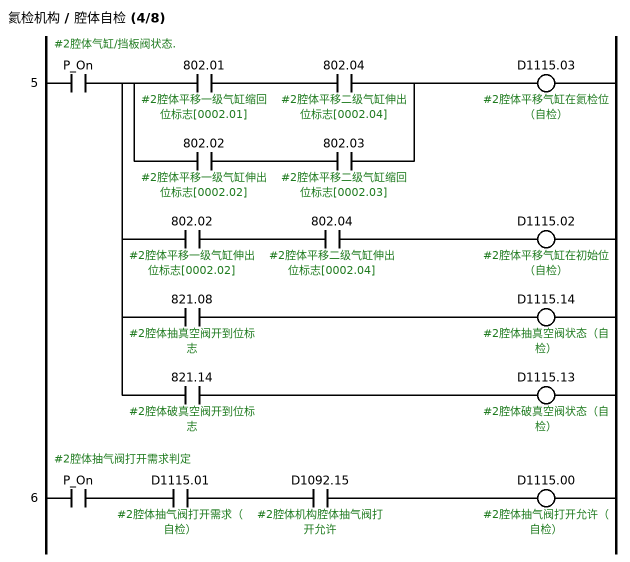
; rung 5: #2腔体气缸/挡板阀状态.
LD P_On
OUT TR0
LD 802.01  ; #2腔体平移一级气缸缩回位标志[0002.01]
AND 802.04  ; #2腔体平移二级气缸伸出位标志[0002.04]
LD 802.02  ; #2腔体平移一级气缸伸出位标志[0002.02]
AND 802.03  ; #2腔体平移二级气缸缩回位标志[0002.03]
ORLD
ANDLD
OUT D1115.03  ; #2腔体平移气缸在氦检位（自检）
LD TR0
AND 802.02  ; #2腔体平移一级气缸伸出位标志[0002.02]
AND 802.04  ; #2腔体平移二级气缸伸出位标志[0002.04]
OUT D1115.02  ; #2腔体平移气缸在初始位（自检）
LD TR0
AND 821.08  ; #2腔体抽真空阀开到位标志
OUT D1115.14  ; #2腔体抽真空阀状态（自检）
LD TR0
AND 821.14  ; #2腔体破真空阀开到位标志
OUT D1115.13  ; #2腔体破真空阀状态（自检）
; rung 6: #2腔体抽气阀打开需求判定
LD P_On
AND D1115.01  ; #2腔体抽气阀打开需求（自检）
AND D1092.15  ; #2腔体机构腔体抽气阀打开允许
OUT D1115.00  ; #2腔体抽气阀打开允许（自检）

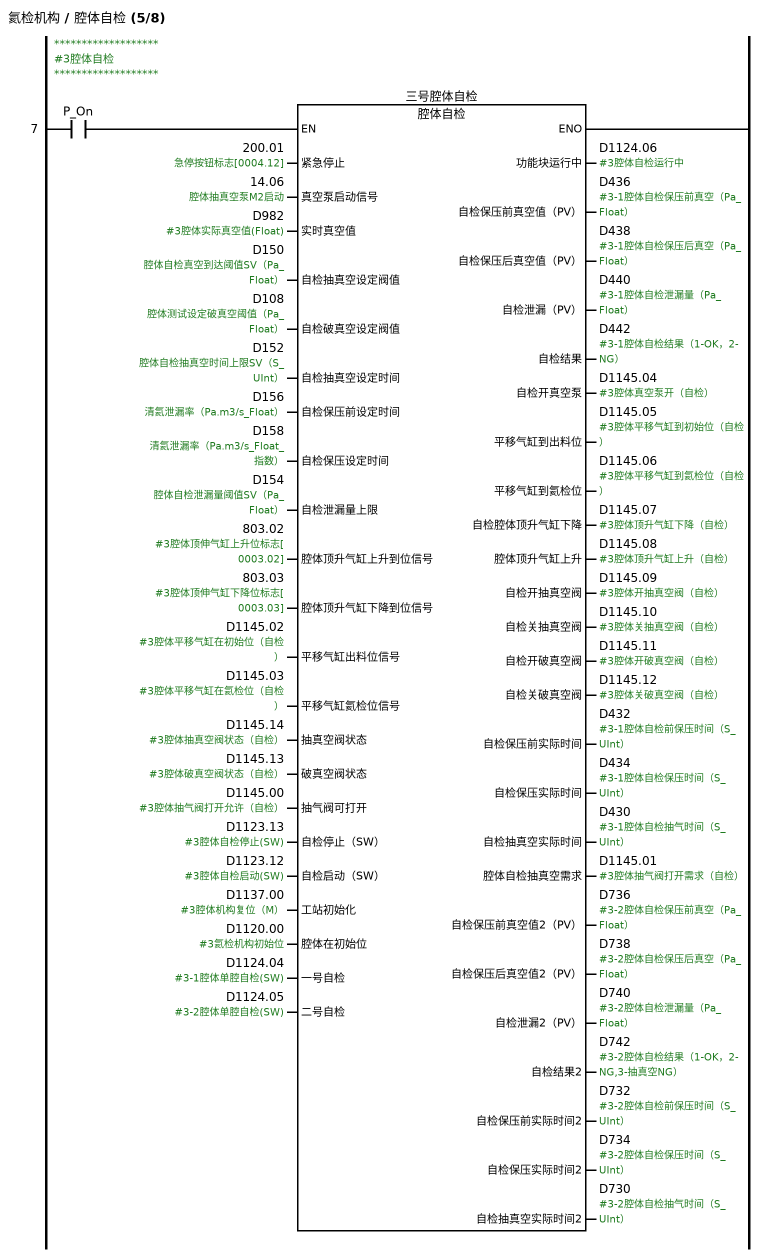
; rung 7: ******************* / #3腔体自检 / *******************
LD P_On
CALL 三号腔体自检 : 腔体自检 (紧急停止 := 200.01, 真空泵启动信号 := 14.06, 实时真空值 := D982, 自检抽真空设定阀值 := D150, 自检破真空设定阀值 := D108, 自检抽真空设定时间 := D152, 自检保压前设定时间 := D156, 自检保压设定时间 := D158, 自检泄漏量上限 := D154, 腔体顶升气缸上升到位信号 := 803.02, 腔体顶升气缸下降到位信号 := 803.03, 平移气缸出料位信号 := D1145.02, 平移气缸氦检位信号 := D1145.03, 抽真空阀状态 := D1145.14, 破真空阀状态 := D1145.13, 抽气阀可打开 := D1145.00, 自检停止（SW） := D1123.13, 自检启动（SW） := D1123.12, 工站初始化 := D1137.00, 腔体在初始位 := D1120.00, 一号自检 := D1124.04, 二号自检 := D1124.05, 功能块运行中 => D1124.06, 自检保压前真空值（PV） => D436, 自检保压后真空值（PV） => D438, 自检泄漏（PV） => D440, 自检结果 => D442, 自检开真空泵 => D1145.04, 平移气缸到出料位 => D1145.05, 平移气缸到氦检位 => D1145.06, 自检腔体顶升气缸下降 => D1145.07, 腔体顶升气缸上升 => D1145.08, 自检开抽真空阀 => D1145.09, 自检关抽真空阀 => D1145.10, 自检开破真空阀 => D1145.11, 自检关破真空阀 => D1145.12, 自检保压前实际时间 => D432, 自检保压实际时间 => D434, 自检抽真空实际时间 => D430, 腔体自检抽真空需求 => D1145.01, 自检保压前真空值2（PV） => D736, 自检保压后真空值2（PV） => D738, 自检泄漏2（PV） => D740, 自检结果2 => D742, 自检保压前实际时间2 => D732, 自检保压实际时间2 => D734, 自检抽真空实际时间2 => D730)  ; 急停按钮标志[0004.12], 腔体抽真空泵M2启动, #3腔体实际真空值(Float), 腔体自检真空到达阈值SV（Pa_Float）, 腔体测试设定破真空阈值（Pa_Float）, 腔体自检抽真空时间上限SV（S_UInt）, 清氦泄漏率（Pa.m3/s_Float）, 清氦泄漏率（Pa.m3/s_Float_指数）, 腔体自检泄漏量阈值SV（Pa_Float）, #3腔体顶伸气缸上升位标志[0003.02], #3腔体顶伸气缸下降位标志[0003.03], #3腔体平移气缸在初始位（自检）, #3腔体平移气缸在氦检位（自检）, #3腔体抽真空阀状态（自检）, #3腔体破真空阀状态（自检）, #3腔体抽气阀打开允许（自检）, #3腔体自检停止(SW), #3腔体自检启动(SW), #3腔体机构复位（M）, #3氦检机构初始位, #3-1腔体单腔自检(SW), #3-2腔体单腔自检(SW), #3腔体自检运行中, #3-1腔体自检保压前真空（Pa_Float）, #3-1腔体自检保压后真空（Pa_Float）, #3-1腔体自检泄漏量（Pa_Float）, #3-1腔体自检结果（1-OK，2-NG）, #3腔体真空泵开（自检）, #3腔体平移气缸到初始位（自检）, #3腔体平移气缸到氦检位（自检）, #3腔体顶升气缸下降（自检）, #3腔体顶升气缸上升（自检）, #3腔体开抽真空阀（自检）, #3腔体关抽真空阀（自检）, #3腔体开破真空阀（自检）, #3腔体关破真空阀（自检）, #3-1腔体自检前保压时间（S_UInt）, #3-1腔体自检保压时间（S_UInt）, #3-1腔体自检抽气时间（S_UInt）, #3腔体抽气阀打开需求（自检）, #3-2腔体自检保压前真空（Pa_Float）, #3-2腔体自检保压后真空（Pa_Float）, #3-2腔体自检泄漏量（Pa_Float）, #3-2腔体自检结果（1-OK，2-NG,3-抽真空NG）, #3-2腔体自检前保压时间（S_UInt）, #3-2腔体自检保压时间（S_UInt）, #3-2腔体自检抽气时间（S_UInt）

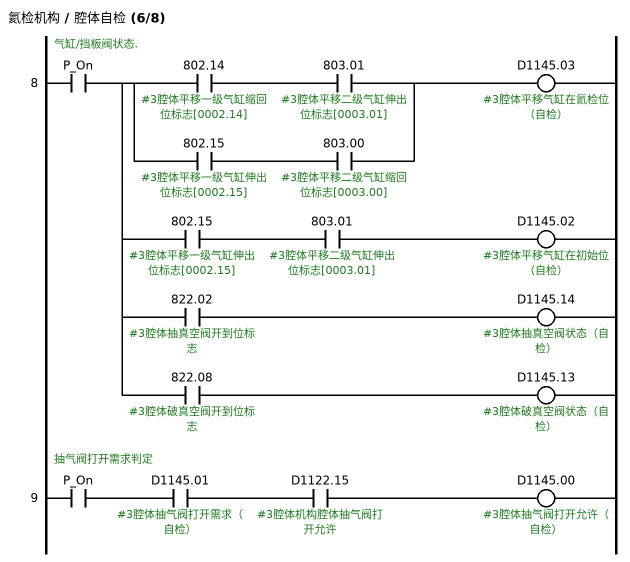
; rung 8: 气缸/挡板阀状态.
LD P_On
OUT TR0
LD 802.14  ; #3腔体平移一级气缸缩回位标志[0002.14]
AND 803.01  ; #3腔体平移二级气缸伸出位标志[0003.01]
LD 802.15  ; #3腔体平移一级气缸伸出位标志[0002.15]
AND 803.00  ; #3腔体平移二级气缸缩回位标志[0003.00]
ORLD
ANDLD
OUT D1145.03  ; #3腔体平移气缸在氦检位（自检）
LD TR0
AND 802.15  ; #3腔体平移一级气缸伸出位标志[0002.15]
AND 803.01  ; #3腔体平移二级气缸伸出位标志[0003.01]
OUT D1145.02  ; #3腔体平移气缸在初始位（自检）
LD TR0
AND 822.02  ; #3腔体抽真空阀开到位标志
OUT D1145.14  ; #3腔体抽真空阀状态（自检）
LD TR0
AND 822.08  ; #3腔体破真空阀开到位标志
OUT D1145.13  ; #3腔体破真空阀状态（自检）
; rung 9: 抽气阀打开需求判定
LD P_On
AND D1145.01  ; #3腔体抽气阀打开需求（自检）
AND D1122.15  ; #3腔体机构腔体抽气阀打开允许
OUT D1145.00  ; #3腔体抽气阀打开允许（自检）

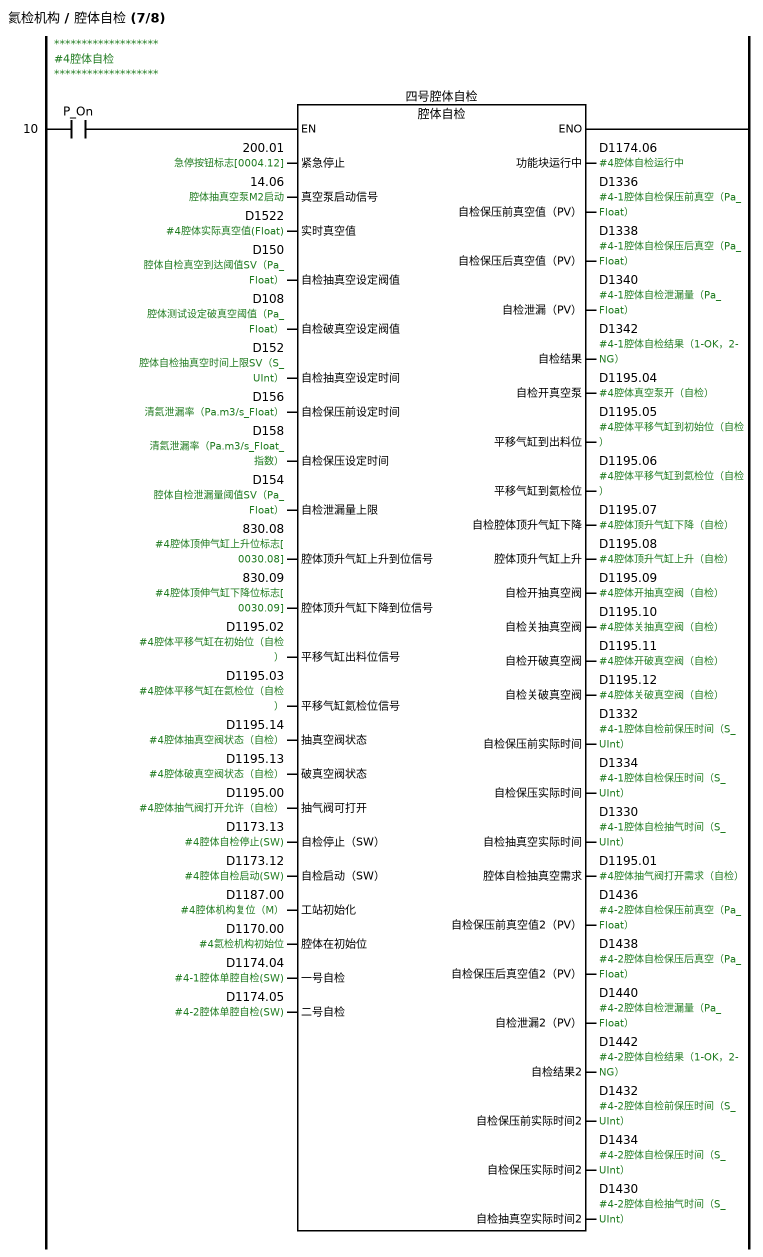
; rung 10: ******************* / #4腔体自检 / *******************
LD P_On
CALL 四号腔体自检 : 腔体自检 (紧急停止 := 200.01, 真空泵启动信号 := 14.06, 实时真空值 := D1522, 自检抽真空设定阀值 := D150, 自检破真空设定阀值 := D108, 自检抽真空设定时间 := D152, 自检保压前设定时间 := D156, 自检保压设定时间 := D158, 自检泄漏量上限 := D154, 腔体顶升气缸上升到位信号 := 830.08, 腔体顶升气缸下降到位信号 := 830.09, 平移气缸出料位信号 := D1195.02, 平移气缸氦检位信号 := D1195.03, 抽真空阀状态 := D1195.14, 破真空阀状态 := D1195.13, 抽气阀可打开 := D1195.00, 自检停止（SW） := D1173.13, 自检启动（SW） := D1173.12, 工站初始化 := D1187.00, 腔体在初始位 := D1170.00, 一号自检 := D1174.04, 二号自检 := D1174.05, 功能块运行中 => D1174.06, 自检保压前真空值（PV） => D1336, 自检保压后真空值（PV） => D1338, 自检泄漏（PV） => D1340, 自检结果 => D1342, 自检开真空泵 => D1195.04, 平移气缸到出料位 => D1195.05, 平移气缸到氦检位 => D1195.06, 自检腔体顶升气缸下降 => D1195.07, 腔体顶升气缸上升 => D1195.08, 自检开抽真空阀 => D1195.09, 自检关抽真空阀 => D1195.10, 自检开破真空阀 => D1195.11, 自检关破真空阀 => D1195.12, 自检保压前实际时间 => D1332, 自检保压实际时间 => D1334, 自检抽真空实际时间 => D1330, 腔体自检抽真空需求 => D1195.01, 自检保压前真空值2（PV） => D1436, 自检保压后真空值2（PV） => D1438, 自检泄漏2（PV） => D1440, 自检结果2 => D1442, 自检保压前实际时间2 => D1432, 自检保压实际时间2 => D1434, 自检抽真空实际时间2 => D1430)  ; 急停按钮标志[0004.12], 腔体抽真空泵M2启动, #4腔体实际真空值(Float), 腔体自检真空到达阈值SV（Pa_Float）, 腔体测试设定破真空阈值（Pa_Float）, 腔体自检抽真空时间上限SV（S_UInt）, 清氦泄漏率（Pa.m3/s_Float）, 清氦泄漏率（Pa.m3/s_Float_指数）, 腔体自检泄漏量阈值SV（Pa_Float）, #4腔体顶伸气缸上升位标志[0030.08], #4腔体顶伸气缸下降位标志[0030.09], #4腔体平移气缸在初始位（自检）, #4腔体平移气缸在氦检位（自检）, #4腔体抽真空阀状态（自检）, #4腔体破真空阀状态（自检）, #4腔体抽气阀打开允许（自检）, #4腔体自检停止(SW), #4腔体自检启动(SW), #4腔体机构复位（M）, #4氦检机构初始位, #4-1腔体单腔自检(SW), #4-2腔体单腔自检(SW), #4腔体自检运行中, #4-1腔体自检保压前真空（Pa_Float）, #4-1腔体自检保压后真空（Pa_Float）, #4-1腔体自检泄漏量（Pa_Float）, #4-1腔体自检结果（1-OK，2-NG）, #4腔体真空泵开（自检）, #4腔体平移气缸到初始位（自检）, #4腔体平移气缸到氦检位（自检）, #4腔体顶升气缸下降（自检）, #4腔体顶升气缸上升（自检）, #4腔体开抽真空阀（自检）, #4腔体关抽真空阀（自检）, #4腔体开破真空阀（自检）, #4腔体关破真空阀（自检）, #4-1腔体自检前保压时间（S_UInt）, #4-1腔体自检保压时间（S_UInt）, #4-1腔体自检抽气时间（S_UInt）, #4腔体抽气阀打开需求（自检）, #4-2腔体自检保压前真空（Pa_Float）, #4-2腔体自检保压后真空（Pa_Float）, #4-2腔体自检泄漏量（Pa_Float）, #4-2腔体自检结果（1-OK，2-NG）, #4-2腔体自检前保压时间（S_UInt）, #4-2腔体自检保压时间（S_UInt）, #4-2腔体自检抽气时间（S_UInt）

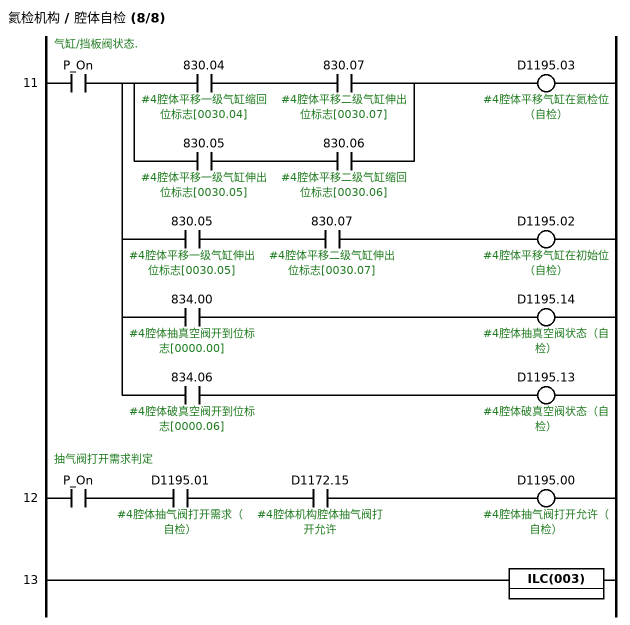
; rung 11: 气缸/挡板阀状态.
LD P_On
OUT TR0
LD 830.04  ; #4腔体平移一级气缸缩回位标志[0030.04]
AND 830.07  ; #4腔体平移二级气缸伸出位标志[0030.07]
LD 830.05  ; #4腔体平移一级气缸伸出位标志[0030.05]
AND 830.06  ; #4腔体平移二级气缸缩回位标志[0030.06]
ORLD
ANDLD
OUT D1195.03  ; #4腔体平移气缸在氦检位（自检）
LD TR0
AND 830.05  ; #4腔体平移一级气缸伸出位标志[0030.05]
AND 830.07  ; #4腔体平移二级气缸伸出位标志[0030.07]
OUT D1195.02  ; #4腔体平移气缸在初始位（自检）
LD TR0
AND 834.00  ; #4腔体抽真空阀开到位标志[0000.00]
OUT D1195.14  ; #4腔体抽真空阀状态（自检）
LD TR0
AND 834.06  ; #4腔体破真空阀开到位标志[0000.06]
OUT D1195.13  ; #4腔体破真空阀状态（自检）
; rung 12: 抽气阀打开需求判定
LD P_On
AND D1195.01  ; #4腔体抽气阀打开需求（自检）
AND D1172.15  ; #4腔体机构腔体抽气阀打开允许
OUT D1195.00  ; #4腔体抽气阀打开允许（自检）
; rung 13
ILC(003)

### Section 指示灯

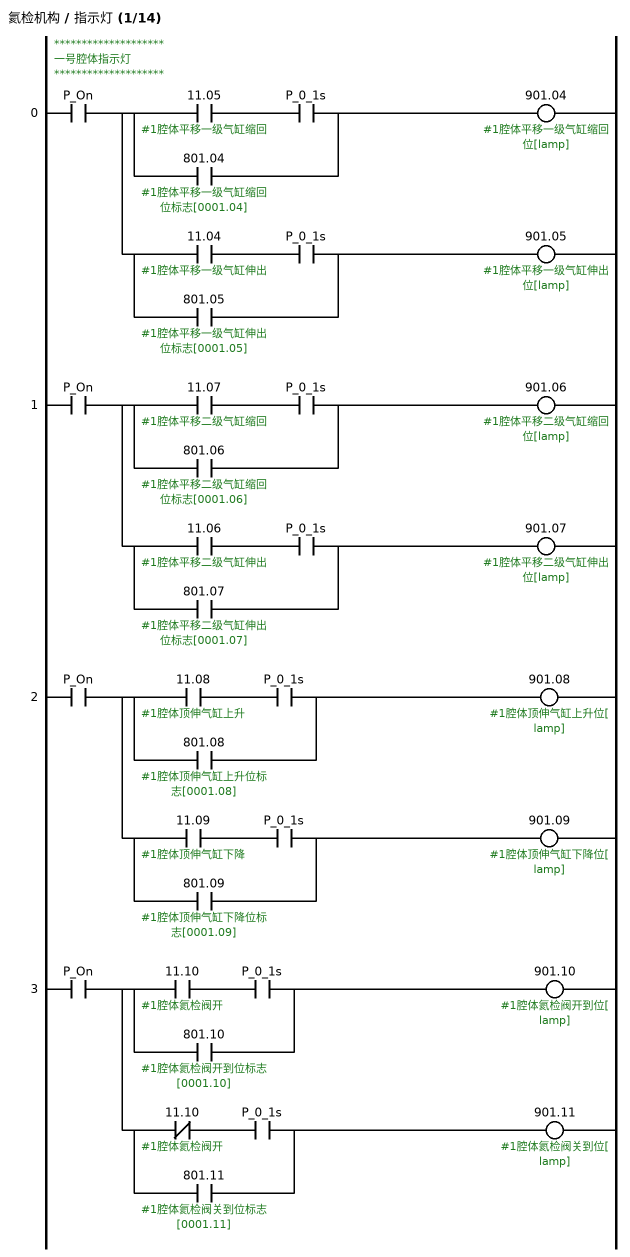
; rung 0: ******************** / 一号腔体指示灯 / ********************
LD P_On
OUT TR0
LD 11.05  ; #1腔体平移一级气缸缩回
AND P_0_1s
OR 801.04  ; #1腔体平移一级气缸缩回位标志[0001.04]
ANDLD
OUT 901.04  ; #1腔体平移一级气缸缩回位[lamp]
LD TR0
LD 11.04  ; #1腔体平移一级气缸伸出
AND P_0_1s
OR 801.05  ; #1腔体平移一级气缸伸出位标志[0001.05]
ANDLD
OUT 901.05  ; #1腔体平移一级气缸伸出位[lamp]
; rung 1
LD P_On
OUT TR0
LD 11.07  ; #1腔体平移二级气缸缩回
AND P_0_1s
OR 801.06  ; #1腔体平移二级气缸缩回位标志[0001.06]
ANDLD
OUT 901.06  ; #1腔体平移二级气缸缩回位[lamp]
LD TR0
LD 11.06  ; #1腔体平移二级气缸伸出
AND P_0_1s
OR 801.07  ; #1腔体平移二级气缸伸出位标志[0001.07]
ANDLD
OUT 901.07  ; #1腔体平移二级气缸伸出位[lamp]
; rung 2
LD P_On
OUT TR0
LD 11.08  ; #1腔体顶伸气缸上升
AND P_0_1s
OR 801.08  ; #1腔体顶伸气缸上升位标志[0001.08]
ANDLD
OUT 901.08  ; #1腔体顶伸气缸上升位[lamp]
LD TR0
LD 11.09  ; #1腔体顶伸气缸下降
AND P_0_1s
OR 801.09  ; #1腔体顶伸气缸下降位标志[0001.09]
ANDLD
OUT 901.09  ; #1腔体顶伸气缸下降位[lamp]
; rung 3
LD P_On
OUT TR0
LD 11.10  ; #1腔体氦检阀开
AND P_0_1s
OR 801.10  ; #1腔体氦检阀开到位标志[0001.10]
ANDLD
OUT 901.10  ; #1腔体氦检阀开到位[lamp]
LD TR0
LDNOT 11.10  ; #1腔体氦检阀开
AND P_0_1s
OR 801.11  ; #1腔体氦检阀关到位标志[0001.11]
ANDLD
OUT 901.11  ; #1腔体氦检阀关到位[lamp]

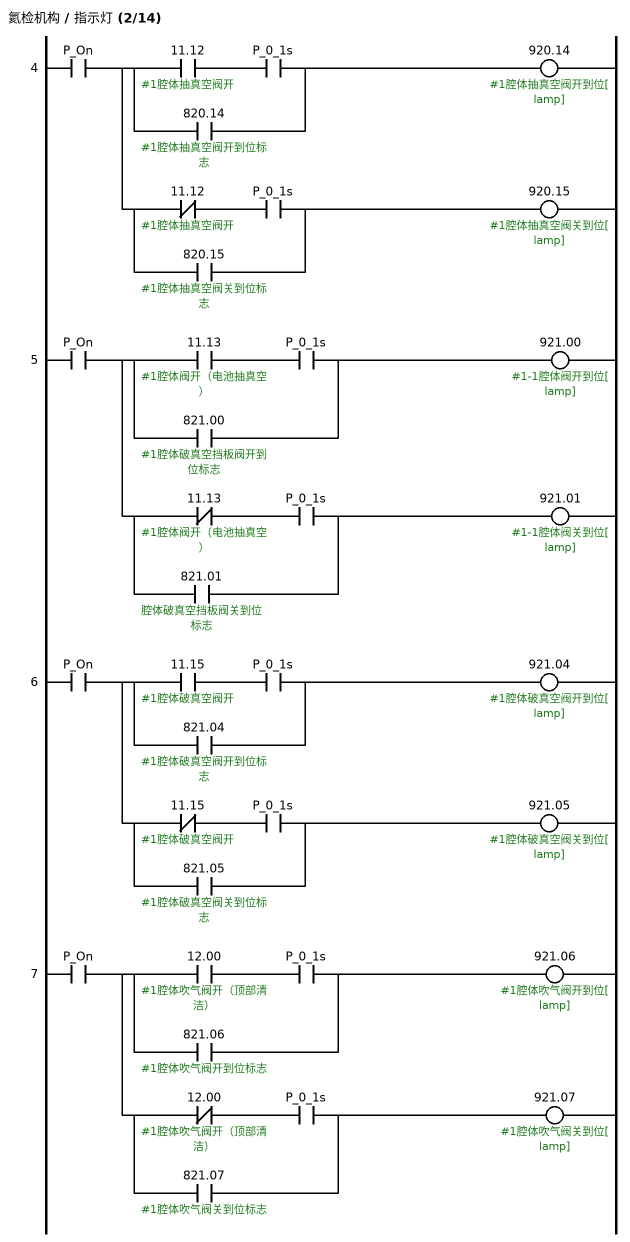
; rung 4
LD P_On
OUT TR0
LD 11.12  ; #1腔体抽真空阀开
AND P_0_1s
OR 820.14  ; #1腔体抽真空阀开到位标志
ANDLD
OUT 920.14  ; #1腔体抽真空阀开到位[lamp]
LD TR0
LDNOT 11.12  ; #1腔体抽真空阀开
AND P_0_1s
OR 820.15  ; #1腔体抽真空阀关到位标志
ANDLD
OUT 920.15  ; #1腔体抽真空阀关到位[lamp]
; rung 5
LD P_On
OUT TR0
LD 11.13  ; #1腔体阀开（电池抽真空）
AND P_0_1s
OR 821.00  ; #1腔体破真空挡板阀开到位标志
ANDLD
OUT 921.00  ; #1-1腔体阀开到位[lamp]
LD TR0
LDNOT 11.13  ; #1腔体阀开（电池抽真空）
AND P_0_1s
OR 821.01  ; 腔体破真空挡板阀关到位标志
ANDLD
OUT 921.01  ; #1-1腔体阀关到位[lamp]
; rung 6
LD P_On
OUT TR0
LD 11.15  ; #1腔体破真空阀开
AND P_0_1s
OR 821.04  ; #1腔体破真空阀开到位标志
ANDLD
OUT 921.04  ; #1腔体破真空阀开到位[lamp]
LD TR0
LDNOT 11.15  ; #1腔体破真空阀开
AND P_0_1s
OR 821.05  ; #1腔体破真空阀关到位标志
ANDLD
OUT 921.05  ; #1腔体破真空阀关到位[lamp]
; rung 7
LD P_On
OUT TR0
LD 12.00  ; #1腔体吹气阀开（顶部清洁）
AND P_0_1s
OR 821.06  ; #1腔体吹气阀开到位标志
ANDLD
OUT 921.06  ; #1腔体吹气阀开到位[lamp]
LD TR0
LDNOT 12.00  ; #1腔体吹气阀开（顶部清洁）
AND P_0_1s
OR 821.07  ; #1腔体吹气阀关到位标志
ANDLD
OUT 921.07  ; #1腔体吹气阀关到位[lamp]

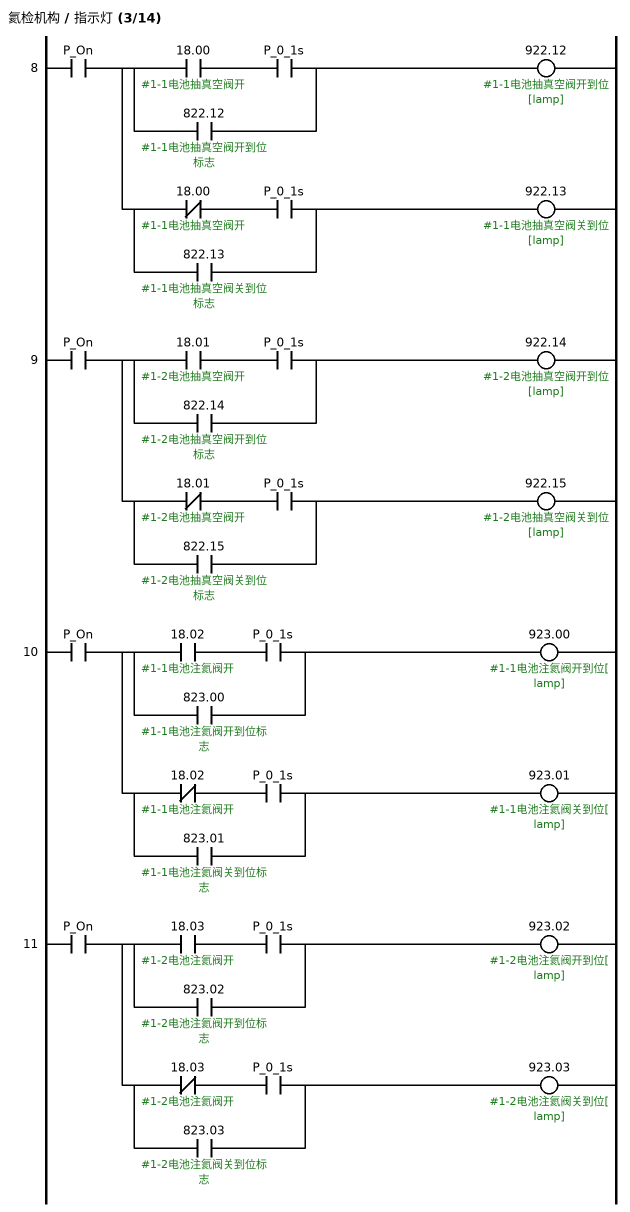
; rung 8
LD P_On
OUT TR0
LD 18.00  ; #1-1电池抽真空阀开
AND P_0_1s
OR 822.12  ; #1-1电池抽真空阀开到位标志
ANDLD
OUT 922.12  ; #1-1电池抽真空阀开到位[lamp]
LD TR0
LDNOT 18.00  ; #1-1电池抽真空阀开
AND P_0_1s
OR 822.13  ; #1-1电池抽真空阀关到位标志
ANDLD
OUT 922.13  ; #1-1电池抽真空阀关到位[lamp]
; rung 9
LD P_On
OUT TR0
LD 18.01  ; #1-2电池抽真空阀开
AND P_0_1s
OR 822.14  ; #1-2电池抽真空阀开到位标志
ANDLD
OUT 922.14  ; #1-2电池抽真空阀开到位[lamp]
LD TR0
LDNOT 18.01  ; #1-2电池抽真空阀开
AND P_0_1s
OR 822.15  ; #1-2电池抽真空阀关到位标志
ANDLD
OUT 922.15  ; #1-2电池抽真空阀关到位[lamp]
; rung 10
LD P_On
OUT TR0
LD 18.02  ; #1-1电池注氦阀开
AND P_0_1s
OR 823.00  ; #1-1电池注氦阀开到位标志
ANDLD
OUT 923.00  ; #1-1电池注氦阀开到位[lamp]
LD TR0
LDNOT 18.02  ; #1-1电池注氦阀开
AND P_0_1s
OR 823.01  ; #1-1电池注氦阀关到位标志
ANDLD
OUT 923.01  ; #1-1电池注氦阀关到位[lamp]
; rung 11
LD P_On
OUT TR0
LD 18.03  ; #1-2电池注氦阀开
AND P_0_1s
OR 823.02  ; #1-2电池注氦阀开到位标志
ANDLD
OUT 923.02  ; #1-2电池注氦阀开到位[lamp]
LD TR0
LDNOT 18.03  ; #1-2电池注氦阀开
AND P_0_1s
OR 823.03  ; #1-2电池注氦阀关到位标志
ANDLD
OUT 923.03  ; #1-2电池注氦阀关到位[lamp]

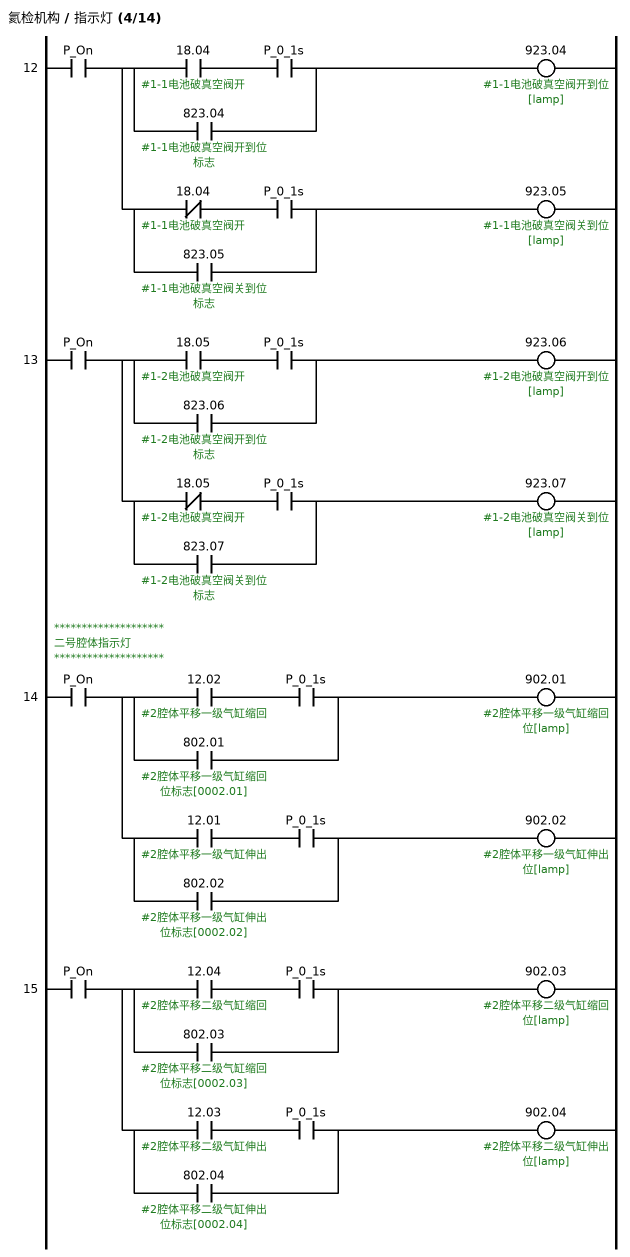
; rung 12
LD P_On
OUT TR0
LD 18.04  ; #1-1电池破真空阀开
AND P_0_1s
OR 823.04  ; #1-1电池破真空阀开到位标志
ANDLD
OUT 923.04  ; #1-1电池破真空阀开到位[lamp]
LD TR0
LDNOT 18.04  ; #1-1电池破真空阀开
AND P_0_1s
OR 823.05  ; #1-1电池破真空阀关到位标志
ANDLD
OUT 923.05  ; #1-1电池破真空阀关到位[lamp]
; rung 13
LD P_On
OUT TR0
LD 18.05  ; #1-2电池破真空阀开
AND P_0_1s
OR 823.06  ; #1-2电池破真空阀开到位标志
ANDLD
OUT 923.06  ; #1-2电池破真空阀开到位[lamp]
LD TR0
LDNOT 18.05  ; #1-2电池破真空阀开
AND P_0_1s
OR 823.07  ; #1-2电池破真空阀关到位标志
ANDLD
OUT 923.07  ; #1-2电池破真空阀关到位[lamp]
; rung 14: ******************** / 二号腔体指示灯 / ********************
LD P_On
OUT TR0
LD 12.02  ; #2腔体平移一级气缸缩回
AND P_0_1s
OR 802.01  ; #2腔体平移一级气缸缩回位标志[0002.01]
ANDLD
OUT 902.01  ; #2腔体平移一级气缸缩回位[lamp]
LD TR0
LD 12.01  ; #2腔体平移一级气缸伸出
AND P_0_1s
OR 802.02  ; #2腔体平移一级气缸伸出位标志[0002.02]
ANDLD
OUT 902.02  ; #2腔体平移一级气缸伸出位[lamp]
; rung 15
LD P_On
OUT TR0
LD 12.04  ; #2腔体平移二级气缸缩回
AND P_0_1s
OR 802.03  ; #2腔体平移二级气缸缩回位标志[0002.03]
ANDLD
OUT 902.03  ; #2腔体平移二级气缸缩回位[lamp]
LD TR0
LD 12.03  ; #2腔体平移二级气缸伸出
AND P_0_1s
OR 802.04  ; #2腔体平移二级气缸伸出位标志[0002.04]
ANDLD
OUT 902.04  ; #2腔体平移二级气缸伸出位[lamp]

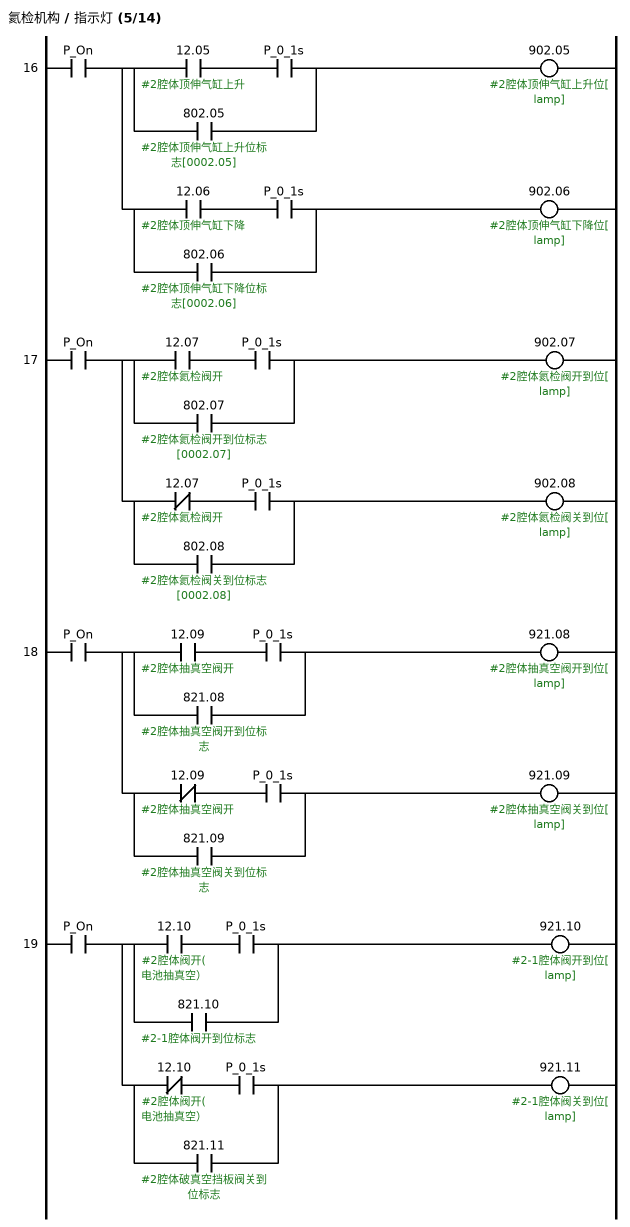
; rung 16
LD P_On
OUT TR0
LD 12.05  ; #2腔体顶伸气缸上升
AND P_0_1s
OR 802.05  ; #2腔体顶伸气缸上升位标志[0002.05]
ANDLD
OUT 902.05  ; #2腔体顶伸气缸上升位[lamp]
LD TR0
LD 12.06  ; #2腔体顶伸气缸下降
AND P_0_1s
OR 802.06  ; #2腔体顶伸气缸下降位标志[0002.06]
ANDLD
OUT 902.06  ; #2腔体顶伸气缸下降位[lamp]
; rung 17
LD P_On
OUT TR0
LD 12.07  ; #2腔体氦检阀开
AND P_0_1s
OR 802.07  ; #2腔体氦检阀开到位标志[0002.07]
ANDLD
OUT 902.07  ; #2腔体氦检阀开到位[lamp]
LD TR0
LDNOT 12.07  ; #2腔体氦检阀开
AND P_0_1s
OR 802.08  ; #2腔体氦检阀关到位标志[0002.08]
ANDLD
OUT 902.08  ; #2腔体氦检阀关到位[lamp]
; rung 18
LD P_On
OUT TR0
LD 12.09  ; #2腔体抽真空阀开
AND P_0_1s
OR 821.08  ; #2腔体抽真空阀开到位标志
ANDLD
OUT 921.08  ; #2腔体抽真空阀开到位[lamp]
LD TR0
LDNOT 12.09  ; #2腔体抽真空阀开
AND P_0_1s
OR 821.09  ; #2腔体抽真空阀关到位标志
ANDLD
OUT 921.09  ; #2腔体抽真空阀关到位[lamp]
; rung 19
LD P_On
OUT TR0
LD 12.10  ; #2腔体阀开(电池抽真空）
AND P_0_1s
OR 821.10  ; #2-1腔体阀开到位标志
ANDLD
OUT 921.10  ; #2-1腔体阀开到位[lamp]
LD TR0
LDNOT 12.10  ; #2腔体阀开(电池抽真空）
AND P_0_1s
OR 821.11  ; #2腔体破真空挡板阀关到位标志
ANDLD
OUT 921.11  ; #2-1腔体阀关到位[lamp]

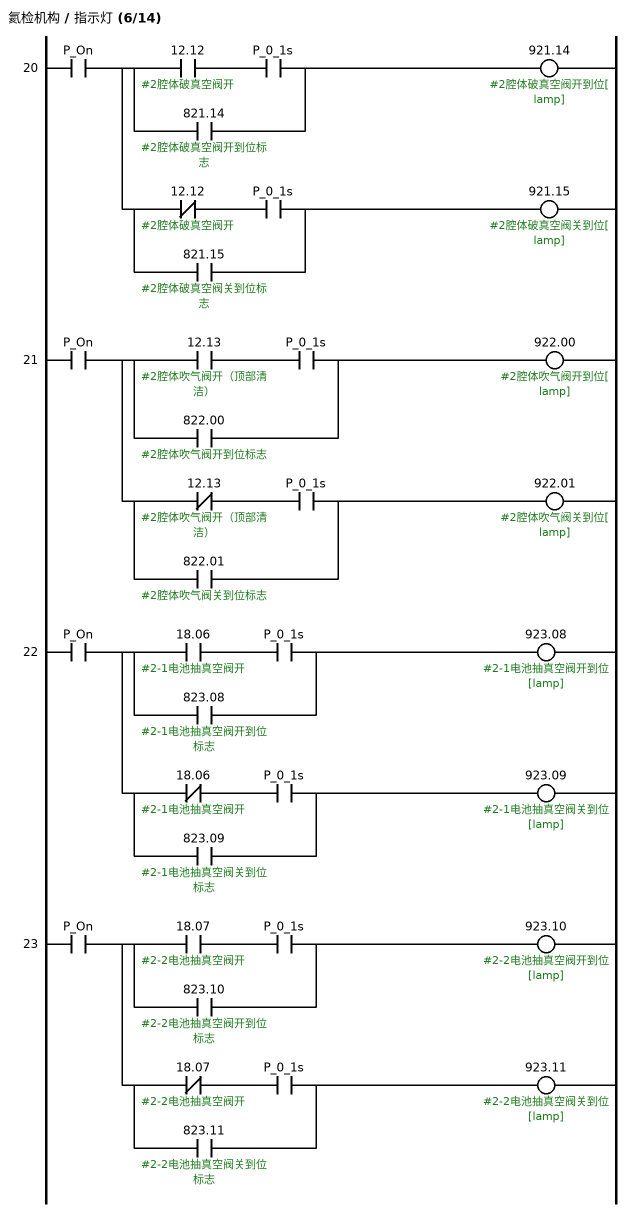
; rung 20
LD P_On
OUT TR0
LD 12.12  ; #2腔体破真空阀开
AND P_0_1s
OR 821.14  ; #2腔体破真空阀开到位标志
ANDLD
OUT 921.14  ; #2腔体破真空阀开到位[lamp]
LD TR0
LDNOT 12.12  ; #2腔体破真空阀开
AND P_0_1s
OR 821.15  ; #2腔体破真空阀关到位标志
ANDLD
OUT 921.15  ; #2腔体破真空阀关到位[lamp]
; rung 21
LD P_On
OUT TR0
LD 12.13  ; #2腔体吹气阀开（顶部清洁）
AND P_0_1s
OR 822.00  ; #2腔体吹气阀开到位标志
ANDLD
OUT 922.00  ; #2腔体吹气阀开到位[lamp]
LD TR0
LDNOT 12.13  ; #2腔体吹气阀开（顶部清洁）
AND P_0_1s
OR 822.01  ; #2腔体吹气阀关到位标志
ANDLD
OUT 922.01  ; #2腔体吹气阀关到位[lamp]
; rung 22
LD P_On
OUT TR0
LD 18.06  ; #2-1电池抽真空阀开
AND P_0_1s
OR 823.08  ; #2-1电池抽真空阀开到位标志
ANDLD
OUT 923.08  ; #2-1电池抽真空阀开到位[lamp]
LD TR0
LDNOT 18.06  ; #2-1电池抽真空阀开
AND P_0_1s
OR 823.09  ; #2-1电池抽真空阀关到位标志
ANDLD
OUT 923.09  ; #2-1电池抽真空阀关到位[lamp]
; rung 23
LD P_On
OUT TR0
LD 18.07  ; #2-2电池抽真空阀开
AND P_0_1s
OR 823.10  ; #2-2电池抽真空阀开到位标志
ANDLD
OUT 923.10  ; #2-2电池抽真空阀开到位[lamp]
LD TR0
LDNOT 18.07  ; #2-2电池抽真空阀开
AND P_0_1s
OR 823.11  ; #2-2电池抽真空阀关到位标志
ANDLD
OUT 923.11  ; #2-2电池抽真空阀关到位[lamp]

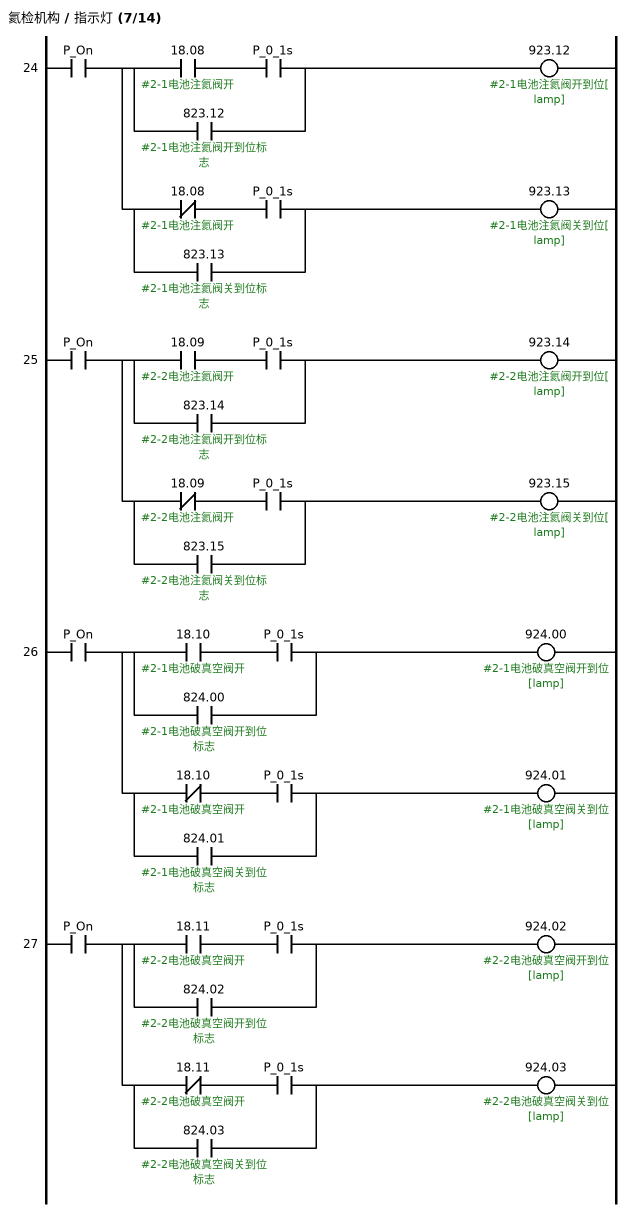
; rung 24
LD P_On
OUT TR0
LD 18.08  ; #2-1电池注氦阀开
AND P_0_1s
OR 823.12  ; #2-1电池注氦阀开到位标志
ANDLD
OUT 923.12  ; #2-1电池注氦阀开到位[lamp]
LD TR0
LDNOT 18.08  ; #2-1电池注氦阀开
AND P_0_1s
OR 823.13  ; #2-1电池注氦阀关到位标志
ANDLD
OUT 923.13  ; #2-1电池注氦阀关到位[lamp]
; rung 25
LD P_On
OUT TR0
LD 18.09  ; #2-2电池注氦阀开
AND P_0_1s
OR 823.14  ; #2-2电池注氦阀开到位标志
ANDLD
OUT 923.14  ; #2-2电池注氦阀开到位[lamp]
LD TR0
LDNOT 18.09  ; #2-2电池注氦阀开
AND P_0_1s
OR 823.15  ; #2-2电池注氦阀关到位标志
ANDLD
OUT 923.15  ; #2-2电池注氦阀关到位[lamp]
; rung 26
LD P_On
OUT TR0
LD 18.10  ; #2-1电池破真空阀开
AND P_0_1s
OR 824.00  ; #2-1电池破真空阀开到位标志
ANDLD
OUT 924.00  ; #2-1电池破真空阀开到位[lamp]
LD TR0
LDNOT 18.10  ; #2-1电池破真空阀开
AND P_0_1s
OR 824.01  ; #2-1电池破真空阀关到位标志
ANDLD
OUT 924.01  ; #2-1电池破真空阀关到位[lamp]
; rung 27
LD P_On
OUT TR0
LD 18.11  ; #2-2电池破真空阀开
AND P_0_1s
OR 824.02  ; #2-2电池破真空阀开到位标志
ANDLD
OUT 924.02  ; #2-2电池破真空阀开到位[lamp]
LD TR0
LDNOT 18.11  ; #2-2电池破真空阀开
AND P_0_1s
OR 824.03  ; #2-2电池破真空阀关到位标志
ANDLD
OUT 924.03  ; #2-2电池破真空阀关到位[lamp]

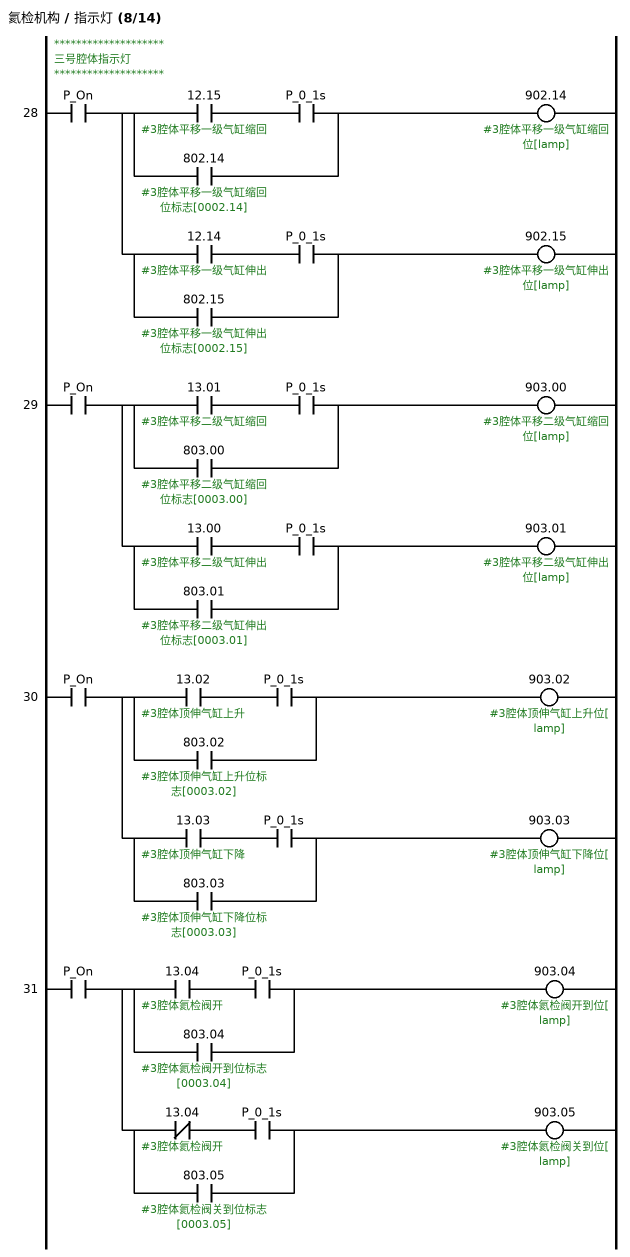
; rung 28: ******************** / 三号腔体指示灯 / ********************
LD P_On
OUT TR0
LD 12.15  ; #3腔体平移一级气缸缩回
AND P_0_1s
OR 802.14  ; #3腔体平移一级气缸缩回位标志[0002.14]
ANDLD
OUT 902.14  ; #3腔体平移一级气缸缩回位[lamp]
LD TR0
LD 12.14  ; #3腔体平移一级气缸伸出
AND P_0_1s
OR 802.15  ; #3腔体平移一级气缸伸出位标志[0002.15]
ANDLD
OUT 902.15  ; #3腔体平移一级气缸伸出位[lamp]
; rung 29
LD P_On
OUT TR0
LD 13.01  ; #3腔体平移二级气缸缩回
AND P_0_1s
OR 803.00  ; #3腔体平移二级气缸缩回位标志[0003.00]
ANDLD
OUT 903.00  ; #3腔体平移二级气缸缩回位[lamp]
LD TR0
LD 13.00  ; #3腔体平移二级气缸伸出
AND P_0_1s
OR 803.01  ; #3腔体平移二级气缸伸出位标志[0003.01]
ANDLD
OUT 903.01  ; #3腔体平移二级气缸伸出位[lamp]
; rung 30
LD P_On
OUT TR0
LD 13.02  ; #3腔体顶伸气缸上升
AND P_0_1s
OR 803.02  ; #3腔体顶伸气缸上升位标志[0003.02]
ANDLD
OUT 903.02  ; #3腔体顶伸气缸上升位[lamp]
LD TR0
LD 13.03  ; #3腔体顶伸气缸下降
AND P_0_1s
OR 803.03  ; #3腔体顶伸气缸下降位标志[0003.03]
ANDLD
OUT 903.03  ; #3腔体顶伸气缸下降位[lamp]
; rung 31
LD P_On
OUT TR0
LD 13.04  ; #3腔体氦检阀开
AND P_0_1s
OR 803.04  ; #3腔体氦检阀开到位标志[0003.04]
ANDLD
OUT 903.04  ; #3腔体氦检阀开到位[lamp]
LD TR0
LDNOT 13.04  ; #3腔体氦检阀开
AND P_0_1s
OR 803.05  ; #3腔体氦检阀关到位标志[0003.05]
ANDLD
OUT 903.05  ; #3腔体氦检阀关到位[lamp]

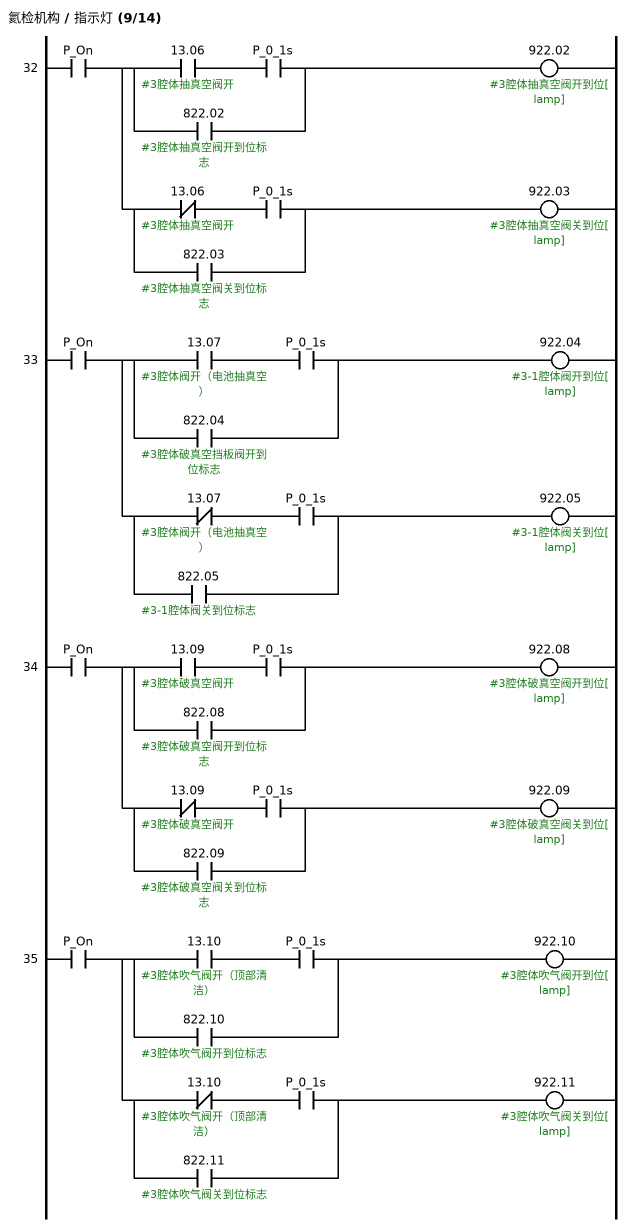
; rung 32
LD P_On
OUT TR0
LD 13.06  ; #3腔体抽真空阀开
AND P_0_1s
OR 822.02  ; #3腔体抽真空阀开到位标志
ANDLD
OUT 922.02  ; #3腔体抽真空阀开到位[lamp]
LD TR0
LDNOT 13.06  ; #3腔体抽真空阀开
AND P_0_1s
OR 822.03  ; #3腔体抽真空阀关到位标志
ANDLD
OUT 922.03  ; #3腔体抽真空阀关到位[lamp]
; rung 33
LD P_On
OUT TR0
LD 13.07  ; #3腔体阀开（电池抽真空）
AND P_0_1s
OR 822.04  ; #3腔体破真空挡板阀开到位标志
ANDLD
OUT 922.04  ; #3-1腔体阀开到位[lamp]
LD TR0
LDNOT 13.07  ; #3腔体阀开（电池抽真空）
AND P_0_1s
OR 822.05  ; #3-1腔体阀关到位标志
ANDLD
OUT 922.05  ; #3-1腔体阀关到位[lamp]
; rung 34
LD P_On
OUT TR0
LD 13.09  ; #3腔体破真空阀开
AND P_0_1s
OR 822.08  ; #3腔体破真空阀开到位标志
ANDLD
OUT 922.08  ; #3腔体破真空阀开到位[lamp]
LD TR0
LDNOT 13.09  ; #3腔体破真空阀开
AND P_0_1s
OR 822.09  ; #3腔体破真空阀关到位标志
ANDLD
OUT 922.09  ; #3腔体破真空阀关到位[lamp]
; rung 35
LD P_On
OUT TR0
LD 13.10  ; #3腔体吹气阀开（顶部清洁）
AND P_0_1s
OR 822.10  ; #3腔体吹气阀开到位标志
ANDLD
OUT 922.10  ; #3腔体吹气阀开到位[lamp]
LD TR0
LDNOT 13.10  ; #3腔体吹气阀开（顶部清洁）
AND P_0_1s
OR 822.11  ; #3腔体吹气阀关到位标志
ANDLD
OUT 922.11  ; #3腔体吹气阀关到位[lamp]

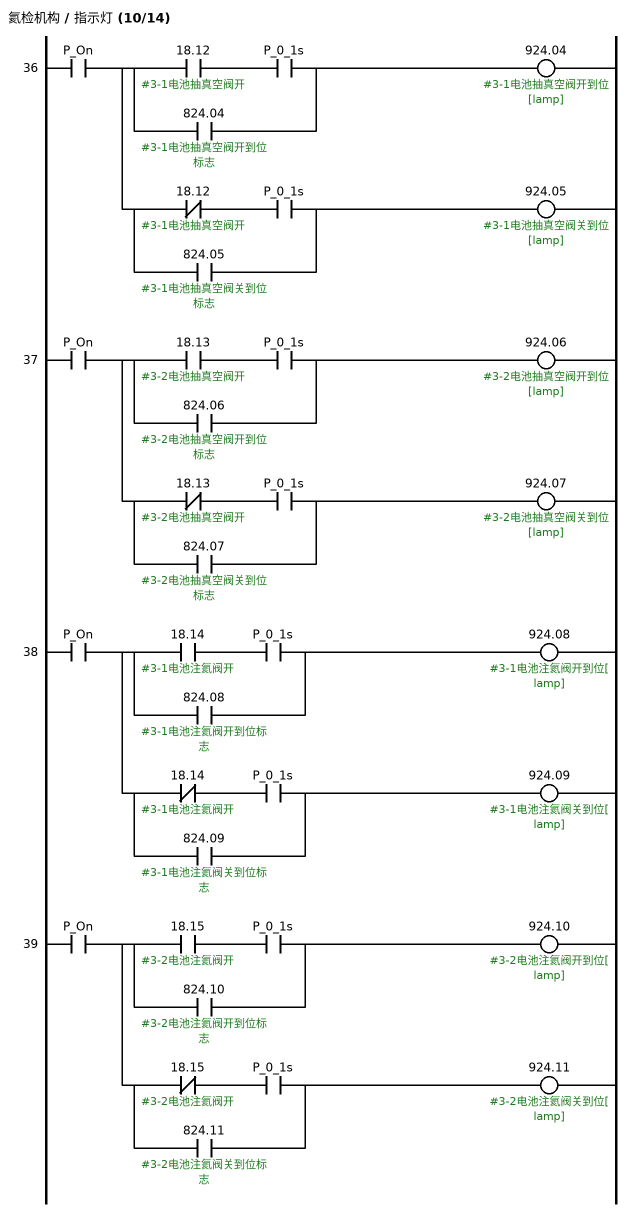
; rung 36
LD P_On
OUT TR0
LD 18.12  ; #3-1电池抽真空阀开
AND P_0_1s
OR 824.04  ; #3-1电池抽真空阀开到位标志
ANDLD
OUT 924.04  ; #3-1电池抽真空阀开到位[lamp]
LD TR0
LDNOT 18.12  ; #3-1电池抽真空阀开
AND P_0_1s
OR 824.05  ; #3-1电池抽真空阀关到位标志
ANDLD
OUT 924.05  ; #3-1电池抽真空阀关到位[lamp]
; rung 37
LD P_On
OUT TR0
LD 18.13  ; #3-2电池抽真空阀开
AND P_0_1s
OR 824.06  ; #3-2电池抽真空阀开到位标志
ANDLD
OUT 924.06  ; #3-2电池抽真空阀开到位[lamp]
LD TR0
LDNOT 18.13  ; #3-2电池抽真空阀开
AND P_0_1s
OR 824.07  ; #3-2电池抽真空阀关到位标志
ANDLD
OUT 924.07  ; #3-2电池抽真空阀关到位[lamp]
; rung 38
LD P_On
OUT TR0
LD 18.14  ; #3-1电池注氦阀开
AND P_0_1s
OR 824.08  ; #3-1电池注氦阀开到位标志
ANDLD
OUT 924.08  ; #3-1电池注氦阀开到位[lamp]
LD TR0
LDNOT 18.14  ; #3-1电池注氦阀开
AND P_0_1s
OR 824.09  ; #3-1电池注氦阀关到位标志
ANDLD
OUT 924.09  ; #3-1电池注氦阀关到位[lamp]
; rung 39
LD P_On
OUT TR0
LD 18.15  ; #3-2电池注氦阀开
AND P_0_1s
OR 824.10  ; #3-2电池注氦阀开到位标志
ANDLD
OUT 924.10  ; #3-2电池注氦阀开到位[lamp]
LD TR0
LDNOT 18.15  ; #3-2电池注氦阀开
AND P_0_1s
OR 824.11  ; #3-2电池注氦阀关到位标志
ANDLD
OUT 924.11  ; #3-2电池注氦阀关到位[lamp]

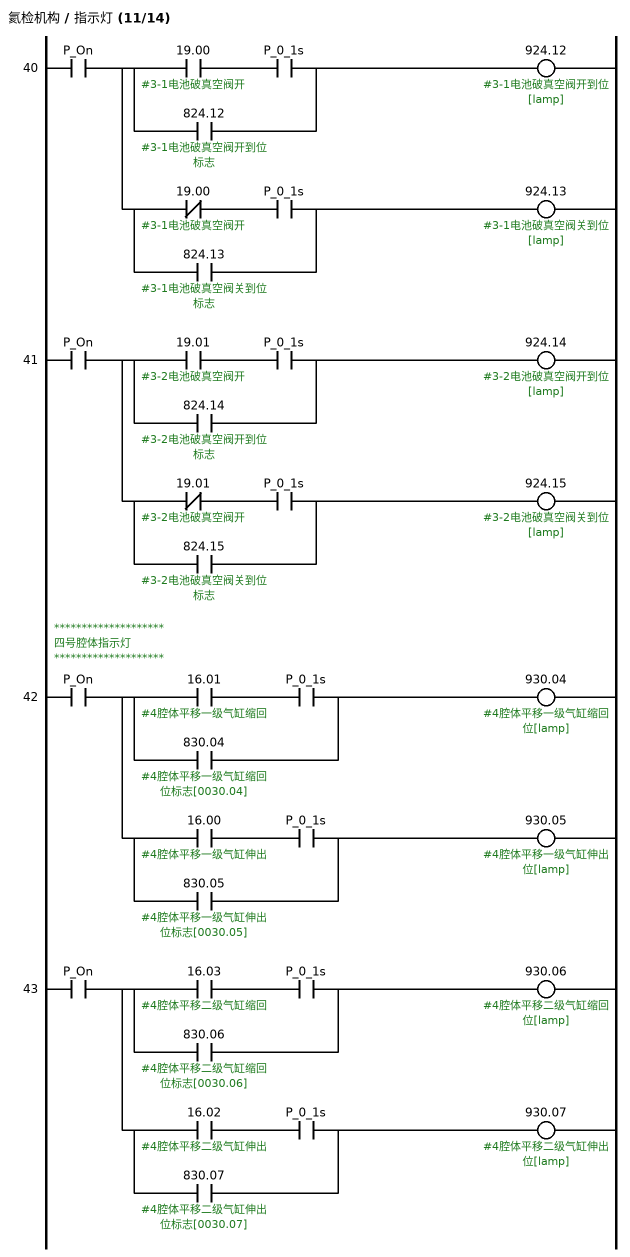
; rung 40
LD P_On
OUT TR0
LD 19.00  ; #3-1电池破真空阀开
AND P_0_1s
OR 824.12  ; #3-1电池破真空阀开到位标志
ANDLD
OUT 924.12  ; #3-1电池破真空阀开到位[lamp]
LD TR0
LDNOT 19.00  ; #3-1电池破真空阀开
AND P_0_1s
OR 824.13  ; #3-1电池破真空阀关到位标志
ANDLD
OUT 924.13  ; #3-1电池破真空阀关到位[lamp]
; rung 41
LD P_On
OUT TR0
LD 19.01  ; #3-2电池破真空阀开
AND P_0_1s
OR 824.14  ; #3-2电池破真空阀开到位标志
ANDLD
OUT 924.14  ; #3-2电池破真空阀开到位[lamp]
LD TR0
LDNOT 19.01  ; #3-2电池破真空阀开
AND P_0_1s
OR 824.15  ; #3-2电池破真空阀关到位标志
ANDLD
OUT 924.15  ; #3-2电池破真空阀关到位[lamp]
; rung 42: ******************** / 四号腔体指示灯 / ********************
LD P_On
OUT TR0
LD 16.01  ; #4腔体平移一级气缸缩回
AND P_0_1s
OR 830.04  ; #4腔体平移一级气缸缩回位标志[0030.04]
ANDLD
OUT 930.04  ; #4腔体平移一级气缸缩回位[lamp]
LD TR0
LD 16.00  ; #4腔体平移一级气缸伸出
AND P_0_1s
OR 830.05  ; #4腔体平移一级气缸伸出位标志[0030.05]
ANDLD
OUT 930.05  ; #4腔体平移一级气缸伸出位[lamp]
; rung 43
LD P_On
OUT TR0
LD 16.03  ; #4腔体平移二级气缸缩回
AND P_0_1s
OR 830.06  ; #4腔体平移二级气缸缩回位标志[0030.06]
ANDLD
OUT 930.06  ; #4腔体平移二级气缸缩回位[lamp]
LD TR0
LD 16.02  ; #4腔体平移二级气缸伸出
AND P_0_1s
OR 830.07  ; #4腔体平移二级气缸伸出位标志[0030.07]
ANDLD
OUT 930.07  ; #4腔体平移二级气缸伸出位[lamp]

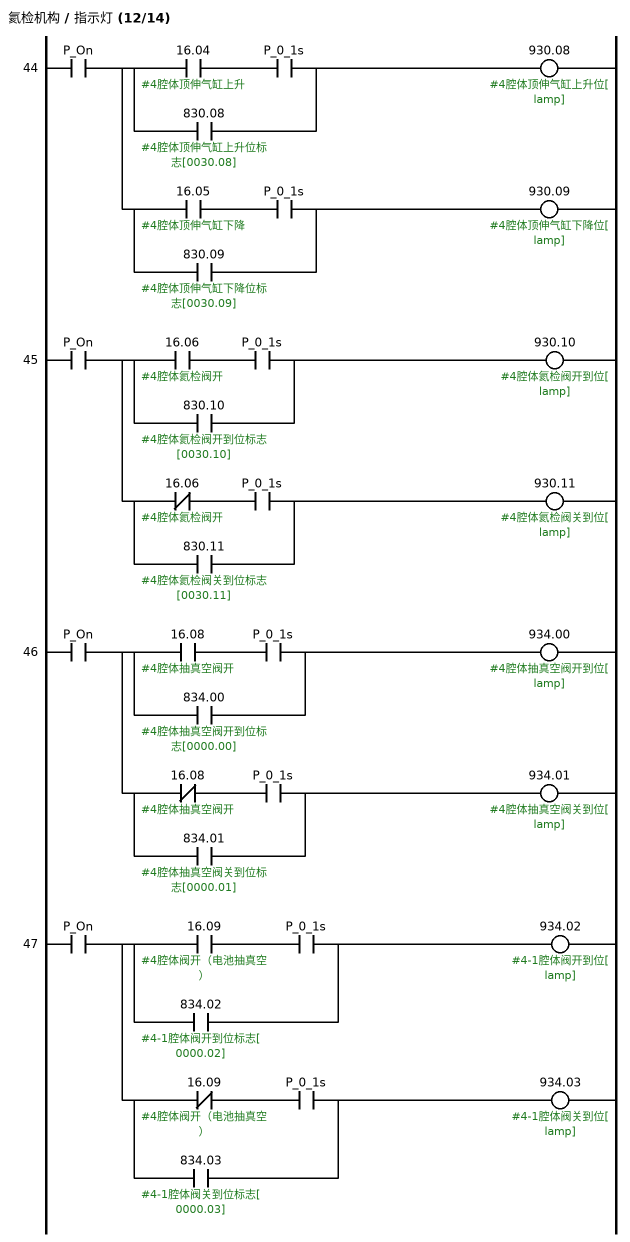
; rung 44
LD P_On
OUT TR0
LD 16.04  ; #4腔体顶伸气缸上升
AND P_0_1s
OR 830.08  ; #4腔体顶伸气缸上升位标志[0030.08]
ANDLD
OUT 930.08  ; #4腔体顶伸气缸上升位[lamp]
LD TR0
LD 16.05  ; #4腔体顶伸气缸下降
AND P_0_1s
OR 830.09  ; #4腔体顶伸气缸下降位标志[0030.09]
ANDLD
OUT 930.09  ; #4腔体顶伸气缸下降位[lamp]
; rung 45
LD P_On
OUT TR0
LD 16.06  ; #4腔体氦检阀开
AND P_0_1s
OR 830.10  ; #4腔体氦检阀开到位标志[0030.10]
ANDLD
OUT 930.10  ; #4腔体氦检阀开到位[lamp]
LD TR0
LDNOT 16.06  ; #4腔体氦检阀开
AND P_0_1s
OR 830.11  ; #4腔体氦检阀关到位标志[0030.11]
ANDLD
OUT 930.11  ; #4腔体氦检阀关到位[lamp]
; rung 46
LD P_On
OUT TR0
LD 16.08  ; #4腔体抽真空阀开
AND P_0_1s
OR 834.00  ; #4腔体抽真空阀开到位标志[0000.00]
ANDLD
OUT 934.00  ; #4腔体抽真空阀开到位[lamp]
LD TR0
LDNOT 16.08  ; #4腔体抽真空阀开
AND P_0_1s
OR 834.01  ; #4腔体抽真空阀关到位标志[0000.01]
ANDLD
OUT 934.01  ; #4腔体抽真空阀关到位[lamp]
; rung 47
LD P_On
OUT TR0
LD 16.09  ; #4腔体阀开（电池抽真空）
AND P_0_1s
OR 834.02  ; #4-1腔体阀开到位标志[0000.02]
ANDLD
OUT 934.02  ; #4-1腔体阀开到位[lamp]
LD TR0
LDNOT 16.09  ; #4腔体阀开（电池抽真空）
AND P_0_1s
OR 834.03  ; #4-1腔体阀关到位标志[0000.03]
ANDLD
OUT 934.03  ; #4-1腔体阀关到位[lamp]

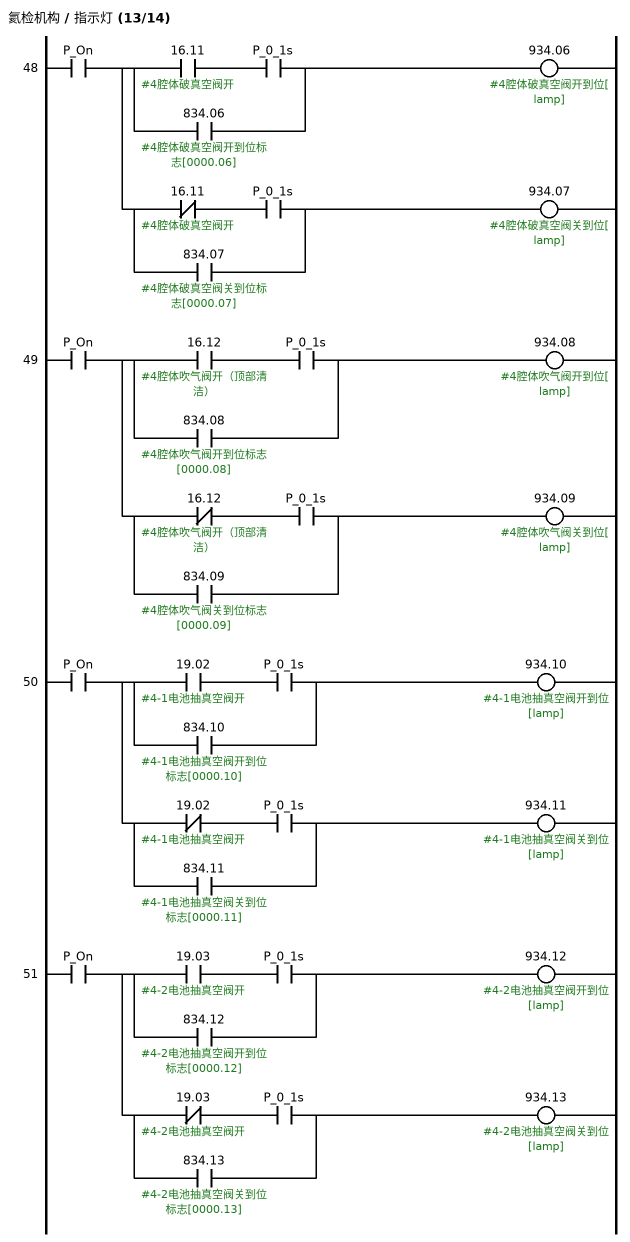
; rung 48
LD P_On
OUT TR0
LD 16.11  ; #4腔体破真空阀开
AND P_0_1s
OR 834.06  ; #4腔体破真空阀开到位标志[0000.06]
ANDLD
OUT 934.06  ; #4腔体破真空阀开到位[lamp]
LD TR0
LDNOT 16.11  ; #4腔体破真空阀开
AND P_0_1s
OR 834.07  ; #4腔体破真空阀关到位标志[0000.07]
ANDLD
OUT 934.07  ; #4腔体破真空阀关到位[lamp]
; rung 49
LD P_On
OUT TR0
LD 16.12  ; #4腔体吹气阀开（顶部清洁）
AND P_0_1s
OR 834.08  ; #4腔体吹气阀开到位标志[0000.08]
ANDLD
OUT 934.08  ; #4腔体吹气阀开到位[lamp]
LD TR0
LDNOT 16.12  ; #4腔体吹气阀开（顶部清洁）
AND P_0_1s
OR 834.09  ; #4腔体吹气阀关到位标志[0000.09]
ANDLD
OUT 934.09  ; #4腔体吹气阀关到位[lamp]
; rung 50
LD P_On
OUT TR0
LD 19.02  ; #4-1电池抽真空阀开
AND P_0_1s
OR 834.10  ; #4-1电池抽真空阀开到位标志[0000.10]
ANDLD
OUT 934.10  ; #4-1电池抽真空阀开到位[lamp]
LD TR0
LDNOT 19.02  ; #4-1电池抽真空阀开
AND P_0_1s
OR 834.11  ; #4-1电池抽真空阀关到位标志[0000.11]
ANDLD
OUT 934.11  ; #4-1电池抽真空阀关到位[lamp]
; rung 51
LD P_On
OUT TR0
LD 19.03  ; #4-2电池抽真空阀开
AND P_0_1s
OR 834.12  ; #4-2电池抽真空阀开到位标志[0000.12]
ANDLD
OUT 934.12  ; #4-2电池抽真空阀开到位[lamp]
LD TR0
LDNOT 19.03  ; #4-2电池抽真空阀开
AND P_0_1s
OR 834.13  ; #4-2电池抽真空阀关到位标志[0000.13]
ANDLD
OUT 934.13  ; #4-2电池抽真空阀关到位[lamp]

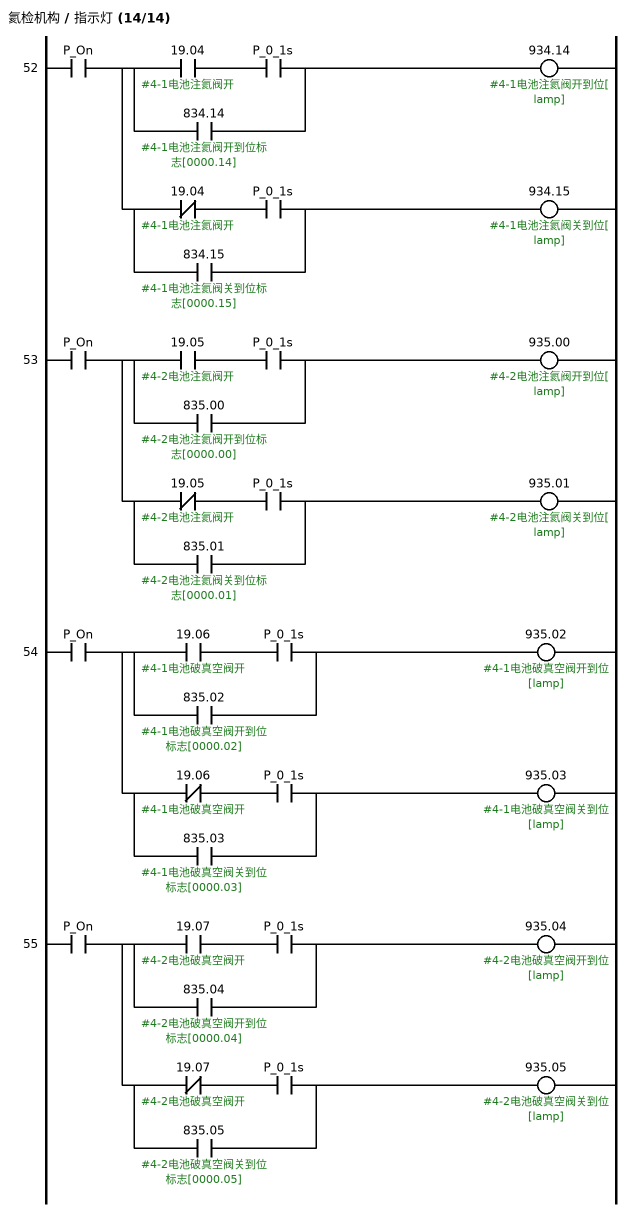
; rung 52
LD P_On
OUT TR0
LD 19.04  ; #4-1电池注氦阀开
AND P_0_1s
OR 834.14  ; #4-1电池注氦阀开到位标志[0000.14]
ANDLD
OUT 934.14  ; #4-1电池注氦阀开到位[lamp]
LD TR0
LDNOT 19.04  ; #4-1电池注氦阀开
AND P_0_1s
OR 834.15  ; #4-1电池注氦阀关到位标志[0000.15]
ANDLD
OUT 934.15  ; #4-1电池注氦阀关到位[lamp]
; rung 53
LD P_On
OUT TR0
LD 19.05  ; #4-2电池注氦阀开
AND P_0_1s
OR 835.00  ; #4-2电池注氦阀开到位标志[0000.00]
ANDLD
OUT 935.00  ; #4-2电池注氦阀开到位[lamp]
LD TR0
LDNOT 19.05  ; #4-2电池注氦阀开
AND P_0_1s
OR 835.01  ; #4-2电池注氦阀关到位标志[0000.01]
ANDLD
OUT 935.01  ; #4-2电池注氦阀关到位[lamp]
; rung 54
LD P_On
OUT TR0
LD 19.06  ; #4-1电池破真空阀开
AND P_0_1s
OR 835.02  ; #4-1电池破真空阀开到位标志[0000.02]
ANDLD
OUT 935.02  ; #4-1电池破真空阀开到位[lamp]
LD TR0
LDNOT 19.06  ; #4-1电池破真空阀开
AND P_0_1s
OR 835.03  ; #4-1电池破真空阀关到位标志[0000.03]
ANDLD
OUT 935.03  ; #4-1电池破真空阀关到位[lamp]
; rung 55
LD P_On
OUT TR0
LD 19.07  ; #4-2电池破真空阀开
AND P_0_1s
OR 835.04  ; #4-2电池破真空阀开到位标志[0000.04]
ANDLD
OUT 935.04  ; #4-2电池破真空阀开到位[lamp]
LD TR0
LDNOT 19.07  ; #4-2电池破真空阀开
AND P_0_1s
OR 835.05  ; #4-2电池破真空阀关到位标志[0000.05]
ANDLD
OUT 935.05  ; #4-2电池破真空阀关到位[lamp]

### Section 外部输出

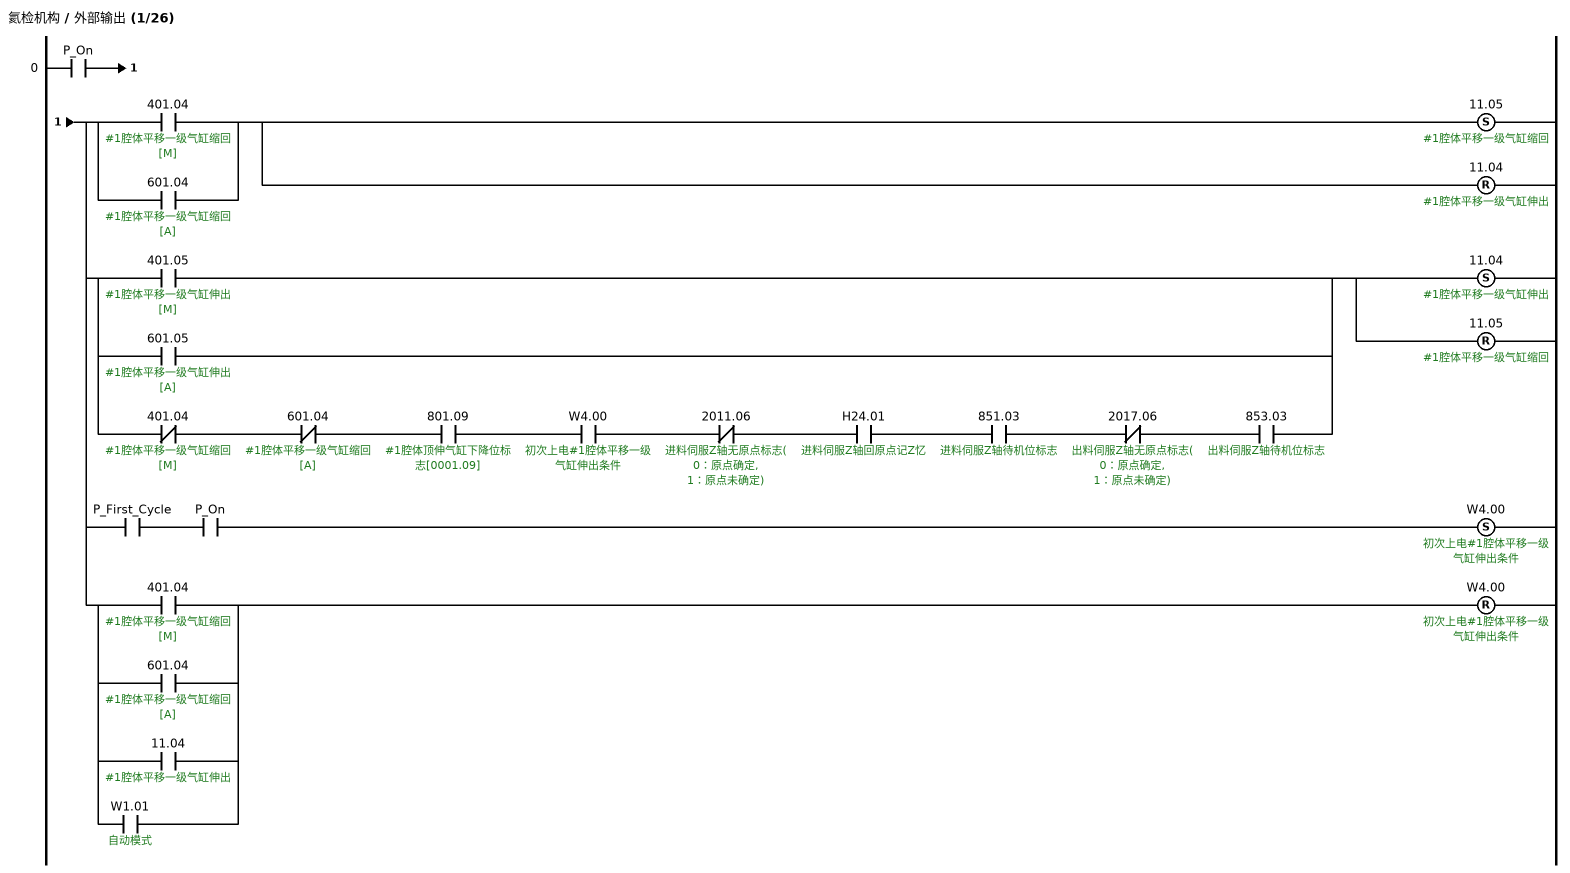
; rung 0
LD P_On
OUT TR0
LD 401.04  ; #1腔体平移一级气缸缩回[M]
OR 601.04  ; #1腔体平移一级气缸缩回[A]
ANDLD
SET 11.05  ; #1腔体平移一级气缸缩回
RSET 11.04  ; #1腔体平移一级气缸伸出
LD TR0
LD 401.05  ; #1腔体平移一级气缸伸出[M]
OR 601.05  ; #1腔体平移一级气缸伸出[A]
LDNOT 401.04  ; #1腔体平移一级气缸缩回[M]
ANDNOT 601.04  ; #1腔体平移一级气缸缩回[A]
AND 801.09  ; #1腔体顶伸气缸下降位标志[0001.09]
AND W4.00  ; 初次上电#1腔体平移一级气缸伸出条件
ANDNOT 2011.06  ; 进料伺服Z轴无原点标志(0：原点确定,1：原点未确定)
AND H24.01  ; 进料伺服Z轴回原点记Z忆
AND 851.03  ; 进料伺服Z轴待机位标志
ANDNOT 2017.06  ; 出料伺服Z轴无原点标志(0：原点确定,1：原点未确定)
AND 853.03  ; 出料伺服Z轴待机位标志
ORLD
ANDLD
SET 11.04  ; #1腔体平移一级气缸伸出
RSET 11.05  ; #1腔体平移一级气缸缩回
LD TR0
AND P_First_Cycle
AND P_On
SET W4.00  ; 初次上电#1腔体平移一级气缸伸出条件
LD TR0
LD 401.04  ; #1腔体平移一级气缸缩回[M]
OR 601.04  ; #1腔体平移一级气缸缩回[A]
OR 11.04  ; #1腔体平移一级气缸伸出
OR W1.01  ; 自动模式
ANDLD
RSET W4.00  ; 初次上电#1腔体平移一级气缸伸出条件

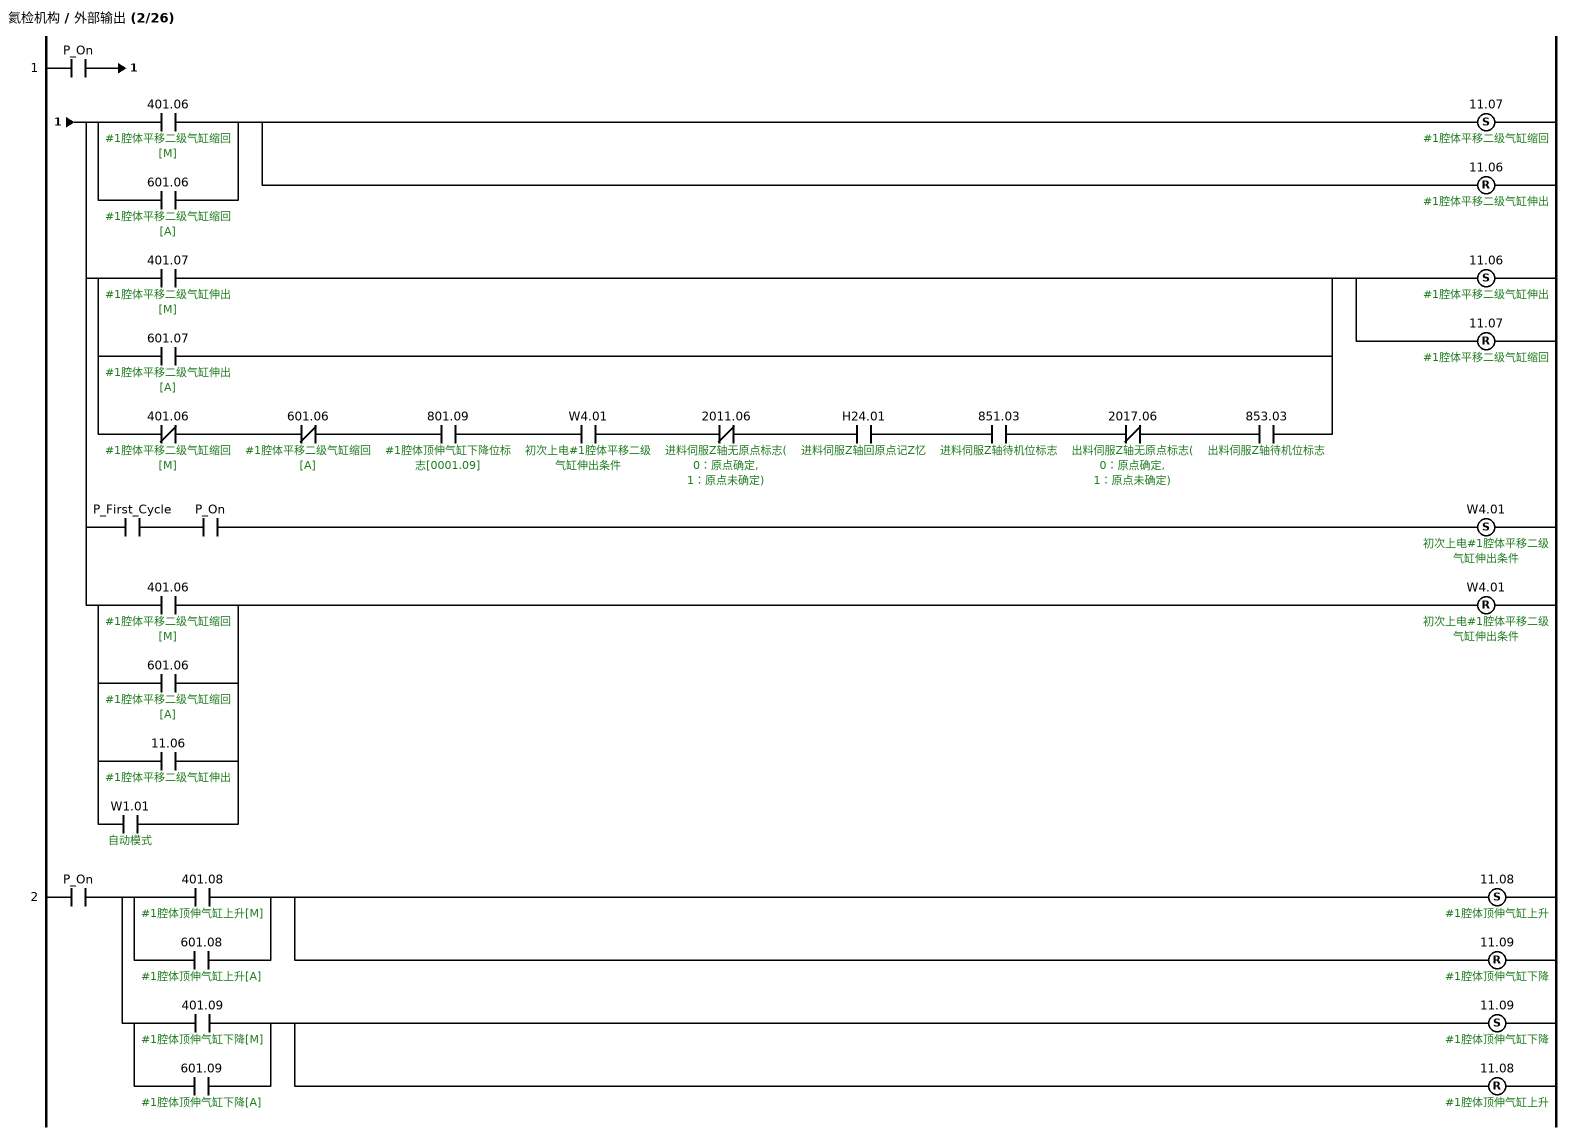
; rung 1
LD P_On
OUT TR0
LD 401.06  ; #1腔体平移二级气缸缩回[M]
OR 601.06  ; #1腔体平移二级气缸缩回[A]
ANDLD
SET 11.07  ; #1腔体平移二级气缸缩回
RSET 11.06  ; #1腔体平移二级气缸伸出
LD TR0
LD 401.07  ; #1腔体平移二级气缸伸出[M]
OR 601.07  ; #1腔体平移二级气缸伸出[A]
LDNOT 401.06  ; #1腔体平移二级气缸缩回[M]
ANDNOT 601.06  ; #1腔体平移二级气缸缩回[A]
AND 801.09  ; #1腔体顶伸气缸下降位标志[0001.09]
AND W4.01  ; 初次上电#1腔体平移二级气缸伸出条件
ANDNOT 2011.06  ; 进料伺服Z轴无原点标志(0：原点确定,1：原点未确定)
AND H24.01  ; 进料伺服Z轴回原点记Z忆
AND 851.03  ; 进料伺服Z轴待机位标志
ANDNOT 2017.06  ; 出料伺服Z轴无原点标志(0：原点确定,1：原点未确定)
AND 853.03  ; 出料伺服Z轴待机位标志
ORLD
ANDLD
SET 11.06  ; #1腔体平移二级气缸伸出
RSET 11.07  ; #1腔体平移二级气缸缩回
LD TR0
AND P_First_Cycle
AND P_On
SET W4.01  ; 初次上电#1腔体平移二级气缸伸出条件
LD TR0
LD 401.06  ; #1腔体平移二级气缸缩回[M]
OR 601.06  ; #1腔体平移二级气缸缩回[A]
OR 11.06  ; #1腔体平移二级气缸伸出
OR W1.01  ; 自动模式
ANDLD
RSET W4.01  ; 初次上电#1腔体平移二级气缸伸出条件
; rung 2
LD P_On
OUT TR0
LD 401.08  ; #1腔体顶伸气缸上升[M]
OR 601.08  ; #1腔体顶伸气缸上升[A]
ANDLD
SET 11.08  ; #1腔体顶伸气缸上升
RSET 11.09  ; #1腔体顶伸气缸下降
LD TR0
LD 401.09  ; #1腔体顶伸气缸下降[M]
OR 601.09  ; #1腔体顶伸气缸下降[A]
ANDLD
SET 11.09  ; #1腔体顶伸气缸下降
RSET 11.08  ; #1腔体顶伸气缸上升

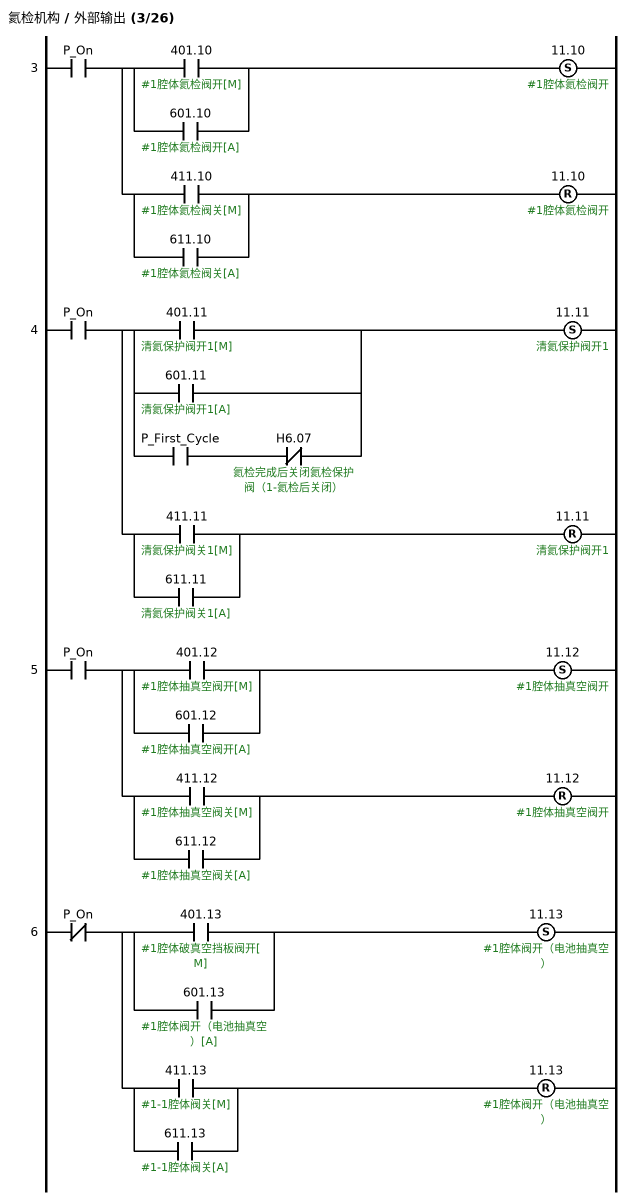
; rung 3
LD P_On
OUT TR0
LD 401.10  ; #1腔体氦检阀开[M]
OR 601.10  ; #1腔体氦检阀开[A]
ANDLD
SET 11.10  ; #1腔体氦检阀开
LD TR0
LD 411.10  ; #1腔体氦检阀关[M]
OR 611.10  ; #1腔体氦检阀关[A]
ANDLD
RSET 11.10  ; #1腔体氦检阀开
; rung 4
LD P_On
OUT TR0
LD 401.11  ; 清氦保护阀开1[M]
OR 601.11  ; 清氦保护阀开1[A]
LD P_First_Cycle  // 保证氦检仪开启时能将管路抽成真空状态
ANDNOT H6.07  ; 氦检完成后关闭氦检保护阀（1-氦检后关闭）
ORLD
ANDLD
SET 11.11  ; 清氦保护阀开1
LD TR0
LD 411.11  ; 清氦保护阀关1[M]
OR 611.11  ; 清氦保护阀关1[A]
ANDLD
RSET 11.11  ; 清氦保护阀开1
; rung 5
LD P_On
OUT TR0
LD 401.12  ; #1腔体抽真空阀开[M]
OR 601.12  ; #1腔体抽真空阀开[A]
ANDLD
SET 11.12  ; #1腔体抽真空阀开
LD TR0
LD 411.12  ; #1腔体抽真空阀关[M]
OR 611.12  ; #1腔体抽真空阀关[A]
ANDLD
RSET 11.12  ; #1腔体抽真空阀开
; rung 6
LDNOT P_On
OUT TR0
LD 401.13  ; #1腔体破真空挡板阀开[M]
OR 601.13  ; #1腔体阀开（电池抽真空）[A]
ANDLD
SET 11.13  ; #1腔体阀开（电池抽真空）
LD TR0
LD 411.13  ; #1-1腔体阀关[M]
OR 611.13  ; #1-1腔体阀关[A]
ANDLD
RSET 11.13  ; #1腔体阀开（电池抽真空）

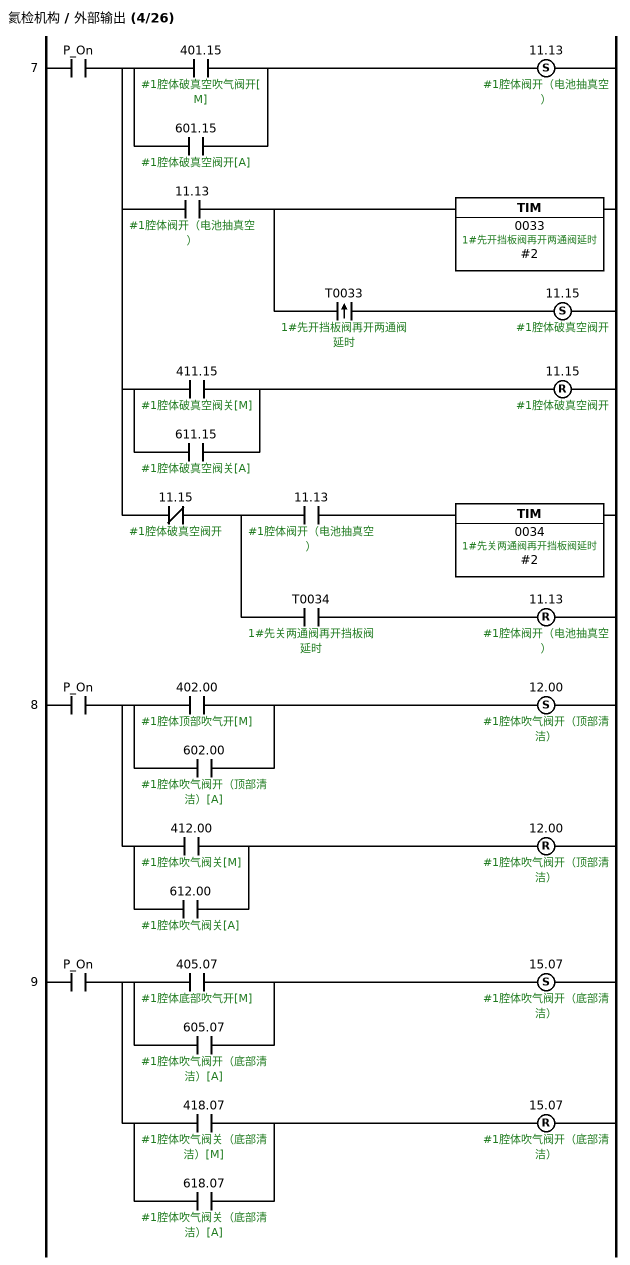
; rung 7
LD P_On
OUT TR0
LD 401.15  ; #1腔体破真空吹气阀开[M]
OR 601.15  ; #1腔体破真空阀开[A]
ANDLD
SET 11.13  ; #1腔体阀开（电池抽真空）
LD TR0
AND 11.13  ; #1腔体阀开（电池抽真空）
TIM 0033 #2  ; 1#先开挡板阀再开两通阀延时
@AND T0033  ; 1#先开挡板阀再开两通阀延时
SET 11.15  ; #1腔体破真空阀开
LD TR0
LD 411.15  ; #1腔体破真空阀关[M]
OR 611.15  ; #1腔体破真空阀关[A]
ANDLD
RSET 11.15  ; #1腔体破真空阀开
LD TR0
ANDNOT 11.15  ; #1腔体破真空阀开
OUT TR0
AND 11.13  ; #1腔体阀开（电池抽真空）
TIM 0034 #2  ; 1#先关两通阀再开挡板阀延时
LD TR0
AND T0034  ; 1#先关两通阀再开挡板阀延时
RSET 11.13  ; #1腔体阀开（电池抽真空）
; rung 8
LD P_On
OUT TR0
LD 402.00  ; #1腔体顶部吹气开[M]
OR 602.00  ; #1腔体吹气阀开（顶部清洁）[A]
ANDLD
SET 12.00  ; #1腔体吹气阀开（顶部清洁）
LD TR0
LD 412.00  ; #1腔体吹气阀关[M]
OR 612.00  ; #1腔体吹气阀关[A]
ANDLD
RSET 12.00  ; #1腔体吹气阀开（顶部清洁）
; rung 9
LD P_On
OUT TR0
LD 405.07  ; #1腔体底部吹气开[M]
OR 605.07  ; #1腔体吹气阀开（底部清洁）[A]
ANDLD
SET 15.07  ; #1腔体吹气阀开（底部清洁）
LD TR0
LD 418.07  ; #1腔体吹气阀关（底部清洁）[M]
OR 618.07  ; #1腔体吹气阀关（底部清洁）[A]
ANDLD
RSET 15.07  ; #1腔体吹气阀开（底部清洁）

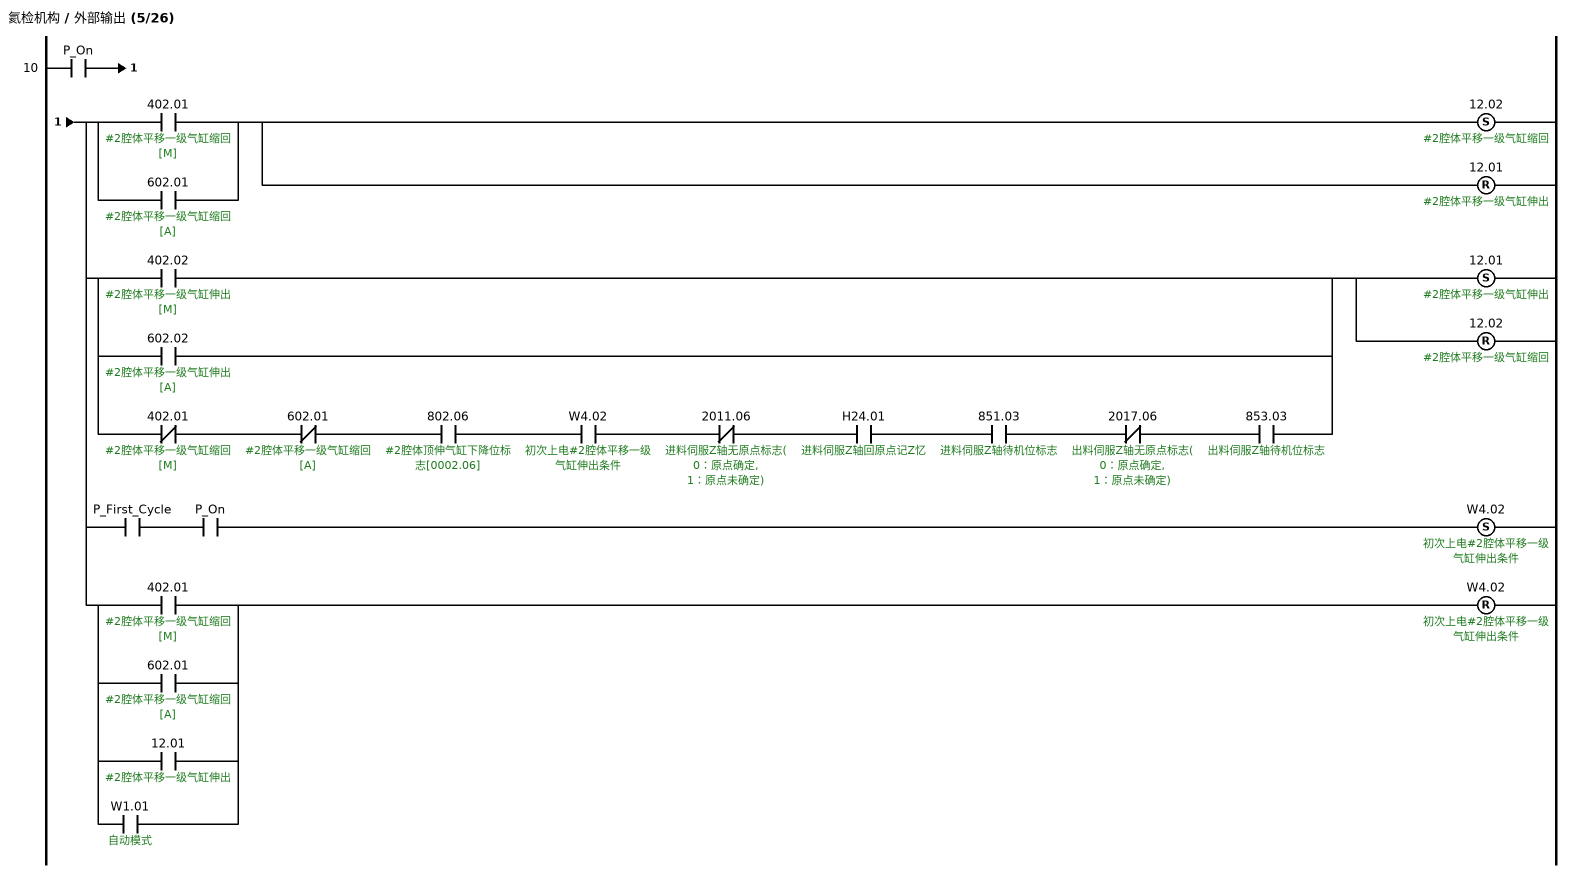
; rung 10
LD P_On
OUT TR0
LD 402.01  ; #2腔体平移一级气缸缩回[M]
OR 602.01  ; #2腔体平移一级气缸缩回[A]
ANDLD
SET 12.02  ; #2腔体平移一级气缸缩回
RSET 12.01  ; #2腔体平移一级气缸伸出
LD TR0
LD 402.02  ; #2腔体平移一级气缸伸出[M]
OR 602.02  ; #2腔体平移一级气缸伸出[A]
LDNOT 402.01  ; #2腔体平移一级气缸缩回[M]
ANDNOT 602.01  ; #2腔体平移一级气缸缩回[A]
AND 802.06  ; #2腔体顶伸气缸下降位标志[0002.06]
AND W4.02  ; 初次上电#2腔体平移一级气缸伸出条件
ANDNOT 2011.06  ; 进料伺服Z轴无原点标志(0：原点确定,1：原点未确定)
AND H24.01  ; 进料伺服Z轴回原点记Z忆
AND 851.03  ; 进料伺服Z轴待机位标志
ANDNOT 2017.06  ; 出料伺服Z轴无原点标志(0：原点确定,1：原点未确定)
AND 853.03  ; 出料伺服Z轴待机位标志
ORLD
ANDLD
SET 12.01  ; #2腔体平移一级气缸伸出
RSET 12.02  ; #2腔体平移一级气缸缩回
LD TR0
AND P_First_Cycle
AND P_On
SET W4.02  ; 初次上电#2腔体平移一级气缸伸出条件
LD TR0
LD 402.01  ; #2腔体平移一级气缸缩回[M]
OR 602.01  ; #2腔体平移一级气缸缩回[A]
OR 12.01  ; #2腔体平移一级气缸伸出
OR W1.01  ; 自动模式
ANDLD
RSET W4.02  ; 初次上电#2腔体平移一级气缸伸出条件

